// TwinCAT 3 PLC project RS485_HausBus
// ProgramVersion: 3.1.4024.0
// libraries:
//   Tc2_SerialCom, * (Beckhoff Automation GmbH)
//   Tc2_Standard, * (Beckhoff Automation GmbH)
//   Tc2_System, * (Beckhoff Automation GmbH)
//   Tc3_Module, * (Beckhoff Automation GmbH)
//   VisuDialogs, * (System)
//   VisuSymbols,3.5.10.0,System
// project tree:
//   DUTs/HausBus/BusTaster/ ST_BusTaster6F_Cnt.TcDUT, ST_BusTaster6F_Input.TcDUT, ST_BusTaster6F_Output.TcDUT
//   DUTs/HausBus/CYD/ ST_BusCYD6F_Input.TcDUT
//   DUTs/HausBus/RelaisModul/ ST_16Relais.TcDUT, ST_BusRelais16F_Cnt.TcDUT, ST_BusRelais16F_Input.TcDUT, ST_BusRelais16F_Output.TcDUT
//   DUTs/HausBus/Service/ ST_FiFoMaster_State.TcDUT, ST_RS485Startup_State.TcDUT (not stored)
//   DUTs/HausBus/ ST_HausBus_Ident.TcDUT
//   / GlobalTextList.TcGTLO, PlcTask.TcTTO, Visualisierungsmanager.TcVMO (not stored)
//   GVLs/ GVL.TcGVL
//   GVLs/RS485_HausBus/ GVL_HausBus_CONSTANT.TcGVL, GVL_HausBus_Devices.TcGVL, GVL_HausBus_Parameter.TcGVL, GVL_RS485FiFoSend.TcGVL, GVL_ServiceVisu.TcGVL
//   POUs/ RS485_COM_PRG.TcPOU
//   POUs/RS485_Hausbus_FB/CYD/ fb_CYDBus6F.TcPOU, fb_StringConvCYDService.TcPOU, fb_StringConvCYDWeb.TcPOU, fb_StringConvCYDWifi.TcPOU
//   POUs/RS485_Hausbus_FB/RS485 COM/FB/ fb_FilterArray.TcPOU
//   POUs/RS485_Hausbus_FB/RS485 COM/ fb_RS485ComCheck.TcPOU, fb_RS485IdScan.TcPOU, fb_RS485Ping.TcPOU
//   POUs/RS485_Hausbus_FB/RS485 COM/RS485_Master/ fb_RS485FiFoMaster.TcPOU, fb_RS485Startup.TcPOU
//   POUs/RS485_Hausbus_FB/BusTaster/ fb_StringConvTB6F.TcPOU, fb_TasterBus6F.TcPOU
//   POUs/RS485_Hausbus_FB/Events/ fb_BusRhdEvent.TcPOU, fb_BusTasterEvent.TcPOU, fb_BusPingEvent.TcPOU, fb_BusTempEvent.TcPOU, fb_BusBrsEvent.TcPOU
//   POUs/RS485_Hausbus_FB/RelaisModul/ fb_RelaisBus16F.TcPOU, fb_StringConvRB16F.TcPOU
//   VISUs/HausBus_RS485/ BusCYD6F_Frame.TcVIS, BusRelais16F_Frame.TcVIS, BusRS485Master_Frame.TcVIS, BusTatster6F_Frame.TcVIS, RS485HB_ServiceVISU.TcVIS
// real-time tasks:
//   TASK PlcTask: cycle T#1ms, priority 20, ADS port 350
// I/O:
//   DEVICE Gerät 2 (EtherCAT), AmsNetId 192.168.178.76.3.1
//     Box 1 (BK1120)
// variable links:
//   RS485_HausBus/RS485_HausBus Instance <-> Device 2 (EtherCAT)/Box 1 (BK1120)
//     PlcTask Inputs/.KL6041In/D[{0..21}] <-> Term 2 (KL6041)/Channel 1/Data In {0..21}  (22 links)
//     PlcTask Inputs/.KL6041In/Status <-> Term 2 (KL6041)/Channel 1/Status
//     PlcTask Inputs/.uiEtherCATStateBK1120_RS485COM <-> InfoData/State
//     PlcTask Inputs/.uiKBusStateBK1120_RS485COM <-> Inputs/CouplerState
//     PlcTask Outputs/.KL6041Out/Ctrl <-> Term 2 (KL6041)/Channel 1/Ctrl
//     PlcTask Outputs/.KL6041Out/D[{0..21}] <-> Term 2 (KL6041)/Channel 1/Data Out {0..21}  (22 links)

CONFIGURATION RS485_HausBus
    RESOURCE PLC ON TwinCAT3
        TASK PlcTask(INTERVAL := T#1ms, PRIORITY := 20);
        PROGRAM RS485_COM_PRG WITH PlcTask : RS485_COM_PRG;
    END_RESOURCE
END_CONFIGURATION

// ---- DUTs/HausBus/BusTaster/ST_BusTaster6F_Cnt.TcDUT
TYPE ST_BusTaster6F_Cnt :
STRUCT
	dwCntButtons    :ARRAY[1..6] OF DWORD;
END_STRUCT
END_TYPE

// ---- DUTs/HausBus/BusTaster/ST_BusTaster6F_Input.TcDUT
TYPE ST_BusTaster6F_Input :
STRUCT
	diID		:DINT;							(* Device ID ( Steht auf dem Aufkleber und wird zur Identifizierung im BUS benötigt)*)
	sName		:STRING;						(* Name des Tasters (zb- Wohnzimmer1 *)
	iLED      	:ARRAY[1..6] OF INT;     	  	(* gewünschter LED-Zustand (TRUE = 100 %)*)
	iLEDExt    	:ARRAY[1..6] OF INT;     	  	(* gewünschter LED-Zustand (TRUE = 100 %)*)
	iLEDBg		:INT;							(* gewünschte Hintergrundbeleuchtung *)
	bReset		:BOOL;							(* Reset des Tasters (Hardware) *)
	bExecute	:BOOL;							(* Aktivierung des Tasters *)
	bExtOutLED	:BOOL;							(* Verwendet die  Extra Ausgänge für LEDs / Mehr Busaulastung!  *)
END_STRUCT
END_TYPE

// ---- DUTs/HausBus/BusTaster/ST_BusTaster6F_Output.TcDUT
TYPE ST_BusTaster6F_Output :
STRUCT
	bButtons    :ARRAY[1..6] OF BOOL;       (*aktueller Tasterstatus (TRUE = gedrückt)*)
	bButtonsExt :ARRAY[1..6] OF BOOL;       (*aktueller Tasterstatus (TRUE = gedrückt)*)
	lrTemp		:LREAL;						(* Temperatur Sensor	*)
	lrRhd		:LREAL;						(* Luftfeuchtigkeit Sensor	*)
	lrBrs		:LREAL;						(* Helligkeit Sensor *)
	
	bCOM			:BOOL;					(*Zeigt die Kommunikation an *)
	bStartupDone	:BOOL;
	
	iState			:BOOL;
	sState			:STRING;
	bError			:BOOL;
END_STRUCT
END_TYPE

// ---- DUTs/HausBus/CYD/ST_BusCYD6F_Input.TcDUT
TYPE ST_BusCYD6F_Input :
STRUCT
	diID			:DINT;							(* Device ID ( Steht auf dem Aufkleber und wird zur Identifizierung im BUS benötigt)*)
	sName			:STRING;						(* Name des Tasters (zb- Wohnzimmer1 *)
	iLED      		:ARRAY[1..6] OF INT;     	  	(* gewünschter LED-Zustand (TRUE = 100 %)*)
	iLEDExt   	 	:ARRAY[1..6] OF INT;     	  	(* gewünschter LED-Zustand (TRUE = 100 %)*)
	iLEDBg			:INT;							(* gewünschte Hintergrundbeleuchtung *)
	
	
	bReset			:BOOL;							(* Reset des Tasters (Hardware) *)
	bExecute		:BOOL;							(* Aktivierung des Tasters *)
	bExtOutLED		:BOOL;							(* Verwendet die  Extra Ausgänge für LEDs / Mehr Busaulastung!  *)
	
	bServiceMode	:BOOL;
	bService		:BOOL;
	bWifi			:BOOL;
	bWebServer		:BOOL;
END_STRUCT
END_TYPE

// ---- DUTs/HausBus/RelaisModul/ST_16Relais.TcDUT
TYPE ST_16Relais :
STRUCT
	bOut	 : ARRAY[1..16] OF BOOL;
END_STRUCT
END_TYPE

// ---- DUTs/HausBus/RelaisModul/ST_BusRelais16F_Cnt.TcDUT
TYPE ST_BusRelais16F_Cnt :
STRUCT
	dwCntRelais    :ARRAY[1..16] OF DWORD;
END_STRUCT
END_TYPE

// ---- DUTs/HausBus/RelaisModul/ST_BusRelais16F_Input.TcDUT
TYPE ST_BusRelais16F_Input :
STRUCT
	diID		:DINT;							(* Device ID ( Steht auf dem Aufkleber und wird zur Identifizierung im BUS benötigt)*)
	sName		:STRING;						(* Name des Tasters (zb- Wohnzimmer1 *)
	bOut     	:ARRAY[1..16] OF BOOL;     	  	(* gewünschter Zustand (TRUE = An%)*)
	bReset		:BOOL;							(* Reset des Tasters (Hardware) *)
	bExecute	:BOOL;							(* Aktivierung des Tasters *)
END_STRUCT
END_TYPE

// ---- DUTs/HausBus/RelaisModul/ST_BusRelais16F_Output.TcDUT
TYPE ST_BusRelais16F_Output :
STRUCT
	bInputs		    :ARRAY[1..8] OF BOOL;       (*aktueller Tasterstatus (TRUE = gedrückt)*)
	bCOM			:BOOL;					(*Zeigt die Kommunikation an *)
	bStartupDone	:BOOL;
	
	iState			:BOOL;
	sState			:STRING;
	bError			:BOOL;
END_STRUCT
END_TYPE

// ---- DUTs/HausBus/Service/ST_FiFoMaster_State.TcDUT
TYPE ST_FiFoMaster_State :
STRUCT
	sReceiveString			:STRING(255);		
	lrBusAuslastung			:LREAL;
	bBusy					:BOOL;
	bDone					:BOOL;
	bError					:BOOL;
	iFiFoCount				:INT;
	iFiFoRow				:INT;
	sSendString				:STRING(255);
	sState					:STRING;
	
END_STRUCT
END_TYPE

// ---- DUTs/HausBus/ST_HausBus_Ident.TcDUT
TYPE ST_HausBus_Ident :
STRUCT
	diID			:DINT;							(* Device ID ( Steht auf dem Aufkleber und wird zur Identifizierung im BUS benötigt)*)
	sName			:STRING;						(* Name des Tasters (zb- Wohnzimmer1 *)	
	sPingIdent		:STRING :='TMP.1.gSTATUS'; 		(* Ping Identifiaktions String, wird bim Pingen gesendet  (Bei Taster = TMP.1.gSTATUS / Relais = OUT.210.rSTATUS / CYD= noch nicht definiert*)
	
END_STRUCT
END_TYPE

// ---- GVLs/GVL.TcGVL
{attribute 'Tc2GvlVarNames'}
VAR_GLOBAL

    KL6041In    					AT %I* : KL6inData22B; // Eingangsdaten von der Klemme
    KL6041Out 						AT %Q* : KL6outData22B; // Ausgangsdaten zur Klemme
	
	uiEtherCATStateBK1120_RS485COM	AT %I* : UINT;			// EtherCAT Status 
	uiKBusStateBK1120_RS485COM		AT %I* : UINT;			// Buskoppler Status
	
	fbTaster 						:ARRAY[1..cMaxBusTaster] OF fb_TasterBus6F;	
	fbRelais						:ARRAY[cMaxBusTaster+1..cMaxBusRelais+cMaxBusTaster+1] OF fb_RelaisBus16F;
END_VAR

// ---- GVLs/RS485_HausBus/GVL_HausBus_CONSTANT.TcGVL
{attribute 'Tc2GvlVarNames'}
VAR_GLOBAL CONSTANT
	cMaxBusTaster			:INT :=10;
	cMaxCYD					:INT :=2;
	cMaxBusRelais			:INT :=1;
	cMaxRS485CMDFiFo		:INT := 15;
	cMaxScanIDs				:INT :=50;
END_VAR

// ---- GVLs/RS485_HausBus/GVL_HausBus_Devices.TcGVL
{attribute 'Tc2GvlVarNames'}
VAR_GLOBAL
	stHBDeviceIdent					:ARRAY[1..cMaxRS485CMDFiFo] OF ST_HausBus_Ident;
	fbTasterHB6F 					:ARRAY[1..cMaxBusTaster] OF fb_TasterBus6F;	
	fbRelaisHB16F					:ARRAY[cMaxBusTaster+1..cMaxBusRelais+cMaxBusTaster+1] OF fb_RelaisBus16F;
	fbCYDHB6F 						:ARRAY[cMaxBusRelais+cMaxBusTaster+2..cMaxBusRelais+cMaxBusTaster+cMaxCYD+1] OF fb_CYDBus6F;	
END_VAR

// ---- GVLs/RS485_HausBus/GVL_HausBus_Parameter.TcGVL
{attribute 'Tc2GvlVarNames'}
VAR_GLOBAL
	
	(* Ping Abfrage *)
	bUseTasterPing						:BOOL := TRUE;			(* Schaltet die Ping empfangsüberprüfung ein um den Verbindungsstatus abzufragen*)
	cTimePingTimeTaster					:TIME := T#40S;			(* Ping Intervallzeit *)	(* Vorerst auf 5min gestellt, da die Taster Automatisch senden (Helligkeit/Luftfeuchtigkeit/Temp usw. *)
	cTimeReceiveTimeoutTaster			:TIME := T#200MS;		(* Ping Empfangs Timeout *)
	
	bUseRelaisPing						:BOOL := TRUE;			(* Schaltet die Ping empfangsüberprüfung ein um den Verbindungsstatus abzufragen*)
	cTimePingTimeRelais					:TIME := T#40S;			(* Ping Intervallzeit *)
	cTimeReceiveTimeoutRelais			:TIME := T#200MS;		(* Ping Empfangs Timeout *)
	
	bUseCYDPing							:BOOL := FALSE;			(* Schaltet die Ping empfangsüberprüfung ein um den Verbindungsstatus abzufragen*)
	cTimePingTimeCYD					:TIME := T#40S;			(* Ping Intervallzeit *)
	cTimeReceiveTimeoutCYD				:TIME := T#200MS;		(* Ping Empfangs Timeout *)
	
	(* FiFo Ping *)
	bUseFiFoPing						:BOOL := TRUE; 			(* Schaltet das Automatische Pingen vom FiFo Master ein, alle Geräte werden von dort aus angepingt *)
	cPingSendTimeFiFo					:TIME := T#19S;			(* Intervall Zeit, wann ein Ping vom FiFo gesendet werden soll an alle Devices *)
	
	(* Nicht verwendet *)
	cMaxPingTry							:INT  := 5;				(* Anzahl der Pingversuche *)
	
END_VAR

// ---- GVLs/RS485_HausBus/GVL_RS485FiFoSend.TcGVL
{attribute 'Tc2GvlVarNames'}
VAR_GLOBAL
	bSendDoneFiFo			:ARRAY[1..cMaxRS485CMDFiFo] OF BOOL;			(* Rückmeldung Aus dem FiFo Master Baustein, dass der Sendevorgang abgeschlossen ist *)
	sSendFiFo				:ARRAY[1..cMaxRS485CMDFiFo] OF STRING(255);		(* Zeile für den FiFo Master Baustein, von jedem einzelnen Busteilnehmer *)
END_VAR

// ---- GVLs/RS485_HausBus/GVL_ServiceVisu.TcGVL
{attribute 'Tc2GvlVarNames'}
VAR_GLOBAL
	iDeviceTasterVisu			:INT := 1;
	iDeviceRelaisVisu			:INT := cMaxBusTaster+1;
	iDeviceCYDVisu				:INT := cMaxBusTaster+cMaxBusRelais+1;
	
	bTasterServiceAktiv			:ARRAY[1..cMaxBusTaster] OF BOOL;
	bRelaisServiceAktiv			:ARRAY[cMaxBusTaster+1..cMaxBusTaster+cMaxBusRelais+1] OF BOOL;
	bCYDServiceAktiv			:ARRAY[cMaxBusRelais+cMaxBusTaster+2..cMaxBusRelais+cMaxBusTaster+cMaxCYD+1] OF BOOL;
	
	stTasterService				:ARRAY[1..cMaxBusTaster] OF ST_BusTaster6F_Input;
	stRelaisService				:ARRAY[cMaxBusTaster+1..cMaxBusTaster+cMaxBusRelais+1] OF ST_BusRelais16F_Input;
	stCYDService				:ARRAY[cMaxBusRelais+cMaxBusTaster+2..cMaxBusRelais+cMaxBusTaster+cMaxCYD+1] OF ST_BusCYD6F_Input;
END_VAR

// ---- POUs/RS485_COM_PRG.TcPOU
(*======================================================================================================================================*)
(*RS485_COM_PRG: Beispielhaftes Programm zum Steuern von HAus-Bus.de Komponenten über RS485 mit TwinCAT
					Achtung dieser POU muss als 1ms Task Aufgerufen werden um Ordnungsgemäß zu laufen *)
(*
Date          	| Version    	| created under        	| Author          	| Remark *)
(*====================================================================================================================================================*)
(*15/05/2025   	| 1.00      		| TC3		  		| N.Kersting       | first release *)
(*====================================================================================================================================================*)

PROGRAM RS485_COM_PRG
VAR  
     i,h,j						:INT;
	
	fbRS485Startup				:fb_RS485Startup;		(* Startup Parametrierung der Klemme/ RS485 Bus *)
	fbRS485SendCmdFiFo			:fb_RS485FiFoMaster;	(* Sende und Empfangs FiFo für RS485 *)
	fbLineControl 				:SerialLineControl;		(* Hält die Serielle Kommunikation Aufrecht *)
	
	fComBufferReset				:ClearComBuffer;		(* Löschen des SPS Internen Bufferinhalts *)
	
	rxBuffer 					:ComBuffer;				(* COM Buffer Empfangen *)
    txBuffer 					:ComBuffer;				(* COM Buffer Senden *)
	
	
END_VAR

(* IDs Setzen *)
ac00_HausBusIdRS485COM();
(* RS485 Klemmen Config *)
ac01_StartupRS485COM();

ACTION ac00_HausBusIdRS485COM:
(* Initialisierung der Gerätenamen *)
(* Achtung nur Beispiele *)
stHBDeviceIdent[1].sName	:=			'Wohnzimmer';
stHBDeviceIdent[1].diID	:=				5256;
stHBDeviceIdent[1].sPingIdent :=		'TMP.1.gSTATUS';

stHBDeviceIdent[2].sName	:=			'Test1';
stHBDeviceIdent[2].diID	:=				5269;
stHBDeviceIdent[2].sPingIdent :=		'TMP.1.gSTATUS';

stHBDeviceIdent[3].sName	:=			'Test2';
stHBDeviceIdent[3].diID	:=				1234;
stHBDeviceIdent[3].sPingIdent :=		'TMP.1.gSTATUS';

stHBDeviceIdent[4].sName	:=			'Test3';
stHBDeviceIdent[4].diID	:=				3333;
stHBDeviceIdent[4].sPingIdent :=		'TMP.1.gSTATUS';

stHBDeviceIdent[5].sName	:=			'Test4';
stHBDeviceIdent[5].diID	:=				4444;
stHBDeviceIdent[5].sPingIdent :=		'TMP.1.gSTATUS';

stHBDeviceIdent[6].sName	:=			'';
stHBDeviceIdent[6].diID	:=				0;
stHBDeviceIdent[6].sPingIdent :=		'TMP.1.gSTATUS';

stHBDeviceIdent[7].sName	:=			'';
stHBDeviceIdent[7].diID	:=				0;
stHBDeviceIdent[7].sPingIdent :=		'TMP.1.gSTATUS';

stHBDeviceIdent[8].sName	:=			'';
stHBDeviceIdent[8].diID	:=				0;
stHBDeviceIdent[8].sPingIdent :=		'TMP.1.gSTATUS';

stHBDeviceIdent[9].sName	:=			'';
stHBDeviceIdent[9].diID	:=				0;
stHBDeviceIdent[9].sPingIdent :=		'TMP.1.gSTATUS';

stHBDeviceIdent[10].sName	:=			'';
stHBDeviceIdent[10].diID	:=			0;
stHBDeviceIdent[10].sPingIdent :=		'TMP.1.gSTATUS';

stHBDeviceIdent[11].sName	:=			'Jalousie 1';
stHBDeviceIdent[11].diID	:=			5614;
stHBDeviceIdent[11].sPingIdent :=		'OUT.210.gSTATUS';

stHBDeviceIdent[12].sName	:=			'';
stHBDeviceIdent[12].diID	:=			0;
stHBDeviceIdent[12].sPingIdent :=		'OUT.210.gSTATUS';

stHBDeviceIdent[13].sName	:=			'CYD Test';
stHBDeviceIdent[13].diID	:=			5999;
stHBDeviceIdent[13].sPingIdent :=		'OUT.210.gSTATUS';
END_ACTION

ACTION ac01_StartupRS485COM:

(* Klemmen Startup, inkl Klemmenkonfiguration usw. *)
fbRS485Startup(
	I_bExecute:= 		TRUE, 
	I_bBusOK:= 			uiEtherCATStateBK1120_RS485COM = 8
						AND uiKBusStateBK1120_RS485COM = 0, 
	I_tStartupVerz:= 	T#5S, 
	IQ_InData:= 		KL6041In, 
	IQ_OutData:= 		KL6041Out, 
	Q_sState=> , 
	Q_bStartupDone=> , 
	Q_bError=> );

(* Aktivierung der Linecontrole erst wenn Startup erfolgt *)	
IF fbRS485Startup.Q_bStartupDone
THEN
	fbLineControl(
		Mode := 		ComSerialLineMode_t.SERIALLINEMODE_KL6_22B_STANDARD,
		pComIn := 		ADR(KL6041In),
		pComOut := 		ADR(KL6041Out),
		SizeComIn := 	UINT_TO_INT(SIZEOF(KL6041In)),
		RxBuffer := 	rxBuffer,
		TxBuffer := 	txBuffer );
				
	(* Relais *)
	ac10_HausBusRelaisRS485COM();
	(* Taster *)
	ac10_HausBusTasterRS485COM();
	(* CYD *)
	ac10_HausBusCYDRS485COM();
	
	
	(* Senden FiFo *)			
	fbRS485SendCmdFiFo(
		I_sSendCmdFiFo:= 		GVL_RS485FiFoSend.sSendFiFo, 
		I_stDeviceIdent :=		stHBDeviceIdent,
		I_bAutoPing:= 			bUseFiFoPing, 
		I_tAutoPingTime:= 		cPingSendTimeFiFo,		 
		I_bManuellMode:= 		, 
		I_sSendCmdManuell:= 	, 
		I_bSendManuell:= 		, 
		I_bExecute:= 			TRUE, 
		I_bBusBelastungstest:= 	, 
		I_bReset:= 				, 
		I_sStartZeichen:= 		, 
		I_sEndZeichen:= 		, 
		I_pTxBuffer:= 			ADR(txBuffer), 
		I_pRxBuffer:= 			ADR(rxBuffer), 
		Q_sReceiveString=> , 
		Q_lrBusAuslastung=> , 
		Q_bBusy=> , 
		Q_bDone=> , 
		Q_bError=> , 
		Q_sState=> , 
		Q_stStates=> );
		
ELSE
	(* Com Buffer zum Resetten *)
	fComBufferReset(Buffer:= rxBuffer);
	fComBufferReset(Buffer:= txBuffer);
END_IF
END_ACTION

ACTION ac10_HausBusCYDRS485COM:
(* Bustaster Aufrufe *)
FOR j := cMaxBusRelais+cMaxBusTaster+2 TO cMaxBusRelais+cMaxBusTaster+cMaxCYD+1 BY 1 DO
		
	fbCYDHB6F[j].I_stInput.sName :=	stHBDeviceIdent[j].sName;
	fbCYDHB6F[j].I_stInput.diID	:=	stHBDeviceIdent[j].diID;
	
	IF GVL_ServiceVisu.bCYDServiceAktiv[j]
	THEN
		fbCYDHB6F[j].I_stInput.iLED := GVL_ServiceVisu.stCYDService[j].iLED;
		fbCYDHB6F[j].I_stInput.iLEDBg := GVL_ServiceVisu.stCYDService[j].iLEDBg;
		fbCYDHB6F[j].I_stInput.iLEDExt := GVL_ServiceVisu.stCYDService[j].iLEDExt;
		fbCYDHB6F[j].I_stInput.bReset := GVL_ServiceVisu.stCYDService[j].bReset;
		fbCYDHB6F[j].I_stInput.bServiceMode := GVL_ServiceVisu.stCYDService[j].bServiceMode;
		fbCYDHB6F[j].I_stInput.bService := GVL_ServiceVisu.stCYDService[j].bService;
		fbCYDHB6F[j].I_stInput.bWifi := GVL_ServiceVisu.stCYDService[j].bWifi;
		fbCYDHB6F[j].I_stInput.bWebServer := GVL_ServiceVisu.stCYDService[j].bWebServer;
		
	END_IF
	
	stCYDService[j].sName :=	fbCYDHB6F[j].I_stInput.sName;
	stCYDService[j].diID :=		fbCYDHB6F[j].I_stInput.diID;
	
	fbCYDHB6F[j].I_stInput.bExecute := TRUE;
	fbCYDHB6F[j](
		I_FifoID :=			j,
		I_bPingStart:= 		TRUE , 	(* Taster Verzögert Pingen, damit weniger Busauslastung entsteht *)
		I_StringReceived:=	fbRS485SendCmdFiFo.Q_sReceiveString);
		
	(* Sendebefehle an FiFo Übergeben *)
	GVL_RS485FiFoSend.sSendFiFo[j] :=	fbCYDHB6F[j].Q_sFiFoSend;
END_FOR
END_ACTION

ACTION ac10_HausBusRelaisRS485COM:
(* BusRelais Aufrufe *)
FOR h := cMaxBusTaster +1 TO cMaxBusRelais+cMaxBusTaster+1 BY 1 DO (*cMaxBusTaster+1..cMaxBusRelais+cMaxBusTaster+1*)
		
	fbRelaisHB16F[h].I_stInput.sName :=	stHBDeviceIdent[h].sName;
	fbRelaisHB16F[h].I_stInput.diID	:=	stHBDeviceIdent[h].diID;
	
	IF GVL_ServiceVisu.bRelaisServiceAktiv[h]
	THEN
		fbRelaisHB16F[h].I_stInput.bOut := stRelaisService[h].bOut;
		fbRelaisHB16F[h].I_stInput.bReset := stRelaisService[h].bReset;
	END_IF
	
	stRelaisService[h].sName :=	fbRelaisHB16F[h].I_stInput.sName;
	stRelaisService[h].diID :=	fbRelaisHB16F[h].I_stInput.diID;
	
	fbRelaisHB16F[h].I_stInput.bExecute := TRUE;
	fbRelaisHB16F[h](
		I_FifoID :=			h,
		I_bPingStart:= 		TRUE,	(* Direkt Starten *)
		I_StringReceived:=	fbRS485SendCmdFiFo.Q_sReceiveString);
		
	(* Sendebefehle an FiFo Übergeben *)
	GVL_RS485FiFoSend.sSendFiFo[h] :=	fbRelaisHB16F[h].Q_sFiFoSend;	
END_FOR
END_ACTION

ACTION ac10_HausBusTasterRS485COM:
(* Bustaster Aufrufe *)
FOR i := 1 TO cMaxBusTaster BY 1 DO
			
	fbTasterHB6F[i].I_stInput.sName :=	stHBDeviceIdent[i].sName;
	fbTasterHB6F[i].I_stInput.diID	:=	stHBDeviceIdent[i].diID;
	
	IF GVL_ServiceVisu.bTasterServiceAktiv[i]
	THEN
		fbTasterHB6F[i].I_stInput.iLED := GVL_ServiceVisu.stTasterService[i].iLED;
		fbTasterHB6F[i].I_stInput.iLEDBg := GVL_ServiceVisu.stTasterService[i].iLEDBg;
		fbTasterHB6F[i].I_stInput.iLEDExt := GVL_ServiceVisu.stTasterService[i].iLEDExt;
		fbTasterHB6F[i].I_stInput.bReset := GVL_ServiceVisu.stTasterService[i].bReset;
	END_IF
	
	stTasterService[i].sName :=	fbTasterHB6F[i].I_stInput.sName;
	stTasterService[i].diID :=	fbTasterHB6F[i].I_stInput.diID;
	
	fbTasterHB6F[i].I_stInput.bExecute := TRUE;
	fbTasterHB6F[i](
		I_FifoID :=			i,
		I_bPingStart:= 		TRUE , 	(* Taster Verzögert Pingen, damit weniger Busauslastung entsteht *)
		I_StringReceived:=	fbRS485SendCmdFiFo.Q_sReceiveString);
		
	(* Sendebefehle an FiFo Übergeben *)
	GVL_RS485FiFoSend.sSendFiFo[i] :=	fbTasterHB6F[i].Q_sFiFoSend;
END_FOR
END_ACTION

END_PROGRAM

// ---- POUs/RS485_Hausbus_FB/RS485 COM/RS485_Master/fb_RS485Startup.TcPOU
(*======================================================================================================================================*)
(*fb_RS485Startup:	Einfacher Baustein um die Hardware für die RS485 Haus-Bus vorzubereiten*)
(*
Date          	| Version    	| created under        	| Author          	| Remark *)
(*====================================================================================================================================================*)
(*13/05/2025   	| 1.00      		| TC3		  		| N.Kersting       | first release *)
(*====================================================================================================================================================*)
FUNCTION_BLOCK fb_RS485Startup
VAR_INPUT
	I_bExecute						:BOOL;
	I_bBusOK						:BOOL;
	I_tStartupVerz					:TIME := T#2S;	(* Startup verzögert ausführen *)
END_VAR
VAR_IN_OUT
	IQ_InData	 					:KL6inData22B;
    IQ_OutData						:KL6outData22B;
END_VAR
VAR_OUTPUT
	Q_sState						:STRING;
	Q_bStartupDone					:BOOL;
	Q_bError						:BOOL;
	Q_stStates						:ST_RS485Startup_State;
END_VAR
VAR
	udBaudrate						:UDINT := 57600;
	byDataBits						:BYTE := 8;
	byStopBits						:BYTE := 1;
	
	tonStartupVerz					:ton;
	fbSerialComReset				:ComReset;
	fComBufferReset					:ClearComBuffer;
	fbSerialConfig 					:KL6Configuration;  // Terminal-Konfiguration (Baud, Parität etc.)
	iStepStartup					:INT;
END_VAR

tonStartupVerz(
	PT :=	I_tStartupVerz);
	
CASE iStepStartup OF 
(*=========================================================================*)
0:	IF NOT Q_bError
		AND I_bBusOK
	THEN
		Q_sState := 'INIT';
	ELSIF
		NOT I_bBusOK
	THEN
		Q_bError := TRUE;
		Q_sState := 'Busverbindung nicht Ok';
	END_IF
	
	tonStartupVerz.IN := FALSE;
	
	fbSerialComReset(
		Execute:= 		FALSE);
		
	fbSerialConfig(
		Execute:= 		FALSE);
		
	IF I_bExecute
		AND I_bBusOK
	THEN
		Q_bStartupDone := FALSE;
		iStepStartup := iStepStartup+1;
	END_IF

(*=========================================================================*)
1:	Q_sState := 'Warten auf Verzögerung';
	tonStartupVerz.IN := TRUE; 
	
	IF tonStartupVerz.Q
	THEN
		iStepStartup := iStepStartup+1;
	END_IF
	
(*=========================================================================*)
2:	Q_sState := 'Serielle Klemme Konfigurieren mit Haus-Bus Vorgaben';	
	
	fbSerialConfig(
		Execute:= 		TRUE, 
		Mode:= 			ComSerialLineMode_t.SERIALLINEMODE_KL6_22B_STANDARD,		 
		Baudrate:= 		udBaudrate, 
		NoDatabits:= 	byDataBits, 
		Parity:= 		ComParity_t.PARITY_EVEN,	 
		Stopbits:= 		byStopBits, 
		Handshake:= 	RS485_HALFDUPLEX, 
		ContinousMode:= , 
		pComIn := 		ADR(IQ_InData), 
		pComOut := 		ADR(IQ_OutData), 
		SizeComIn := 	SIZEOF(IQ_InData),
		Done=> , 
		Busy=> , 
		Error=> , 
		ErrorId=> );
	
	IF fbSerialConfig.Done
	THEN
		fbSerialConfig(
			Execute:= 		FALSE); 
			
		iStepStartup := 3;
	ELSIF
		fbSerialConfig.Error
	THEN
		Q_sState := 'Error fbSerialConfig ID: ';
		Q_sState := CONCAT(Q_sState,INT_TO_STRING(fbSerialConfig.ErrorID));
		iStepStartup := -2;	//Error
	END_IF

(*=========================================================================*)
3:	Q_sState := 'Serielle Klemme Reset Auführen';	
		
	fbSerialComReset(
		Execute:= 		TRUE, 
		pComIn := 		ADR(IQ_InData), 
		pComOut := 		ADR(IQ_OutData), 
		SizeComIn := 	SIZEOF(IQ_InData),
		Done=> , 
		Busy=> , 
		Error=> , 
		ErrorID=> );	
		
	IF fbSerialComReset.Done
	THEN
		iStepStartup := 999;
	ELSIF
		fbSerialComReset.Error
	THEN
		Q_sState := 'Error fbSerialComReset ID: ';
		Q_sState := CONCAT(Q_sState,INT_TO_STRING(fbSerialComReset.ErrorID));
		iStepStartup := -3;	//Error
	END_IF
	
(*=========================================================================*)
999:Q_sState := 'Startup Ausgeführt!';	
	Q_bStartupDone := TRUE;
	Q_bError := FALSE;
	
	IF NOT I_bBusOK
	THEN
		Q_bStartupDone := FALSE;
		iStepStartup := 0;
	END_IF

ELSE
	(* ERROR *)
	Q_bError := TRUE;
	iStepStartup := 0;
END_CASE

(* StatusStruktur für Visu *)
Q_stStates.bBusOk				:=	I_bBusOK;
Q_stStates.bStartupDone			:=	Q_bStartupDone;
Q_stStates.bStartupError		:=	Q_bError;
Q_stStates.sStartupState		:=	Q_sState;

END_FUNCTION_BLOCK

// ---- POUs/RS485_Hausbus_FB/RS485 COM/RS485_Master/fb_RS485FiFoMaster.TcPOU
(*======================================================================================================================================*)
(*fb_RS485FiFoMaster:	Einfaches Senden eines Telegrams über RS485*)
(*
Date          	| Version    	| created under        	| Author          	| Remark *)
(*====================================================================================================================================================*)
(*10/05/2025   	| 1.00      		| TC3		  		| N.Kersting       | first release *)
(*10/05/2025   	| 1.01      		| TC3		  		| N.Kersting       | Nun wird der Empfang auch mit Implementiert  *)
(*13/05/2025   	| 1.02      		| TC3		  		| N.Kersting       | Busbelastungstest Implementiert - Sendet Durchgehend Strings *)
(*14/05/2025   	| 1.03      		| TC3		  		| N.Kersting       | Busauslastung direkt Implementiert *)
(*27/05/2025   	| 1.04      		| TC3		  		| N.Kersting       | Neuen Manuell Mode implementiert um einen Manuell generierten String allein zu Senden *)
(*28/05/2025   	| 1.05      		| TC3		  		| N.Kersting       | Neue Automatisch Ping Funktion hinzugefügt & Wichtiger Bugfix *)
(*02/06/2025   	| 2.00      		| TC3		  		| N.Kersting       | Neue Verbesserte Collision Detection, verhindert, dass Senden bei gefülltem Epmfangspuffer *)
(*03/06/2025   	| 2.01      		| TC3		  		| N.Kersting       | Collision Detection nun aufgeeilt in Empfang und Senden *)
(*03/06/2025   	| 2.02      		| TC3		  		| N.Kersting       | Neue Bus Scan Funktion Implementiert, Scannt alle Teilnehmer Ids im Bus (nur im Manuell Mode verfügbar) *)
(*====================================================================================================================================================*)
FUNCTION_BLOCK fb_RS485FiFoMaster
VAR_INPUT
	I_sSendCmdFiFo				:ARRAY[1..cMaxRS485CMDFiFo] OF STRING(255);
	I_stDeviceIdent				:ARRAY[1..cMaxRS485CMDFiFo] OF ST_HausBus_Ident;	(* Um Zyklisch einzelnt anzupingen *)
	
	I_bAutoPing					:BOOL;												(* Wenn Aktiv wird Zyklisch Automatisch ein Ping gesendet, welcher von den einzelnen Kommunikationsbausteinen ausgewertet werden kann *)
	I_tAutoPingTime				:TIME :=T#10S;										(* Die Intervallzeit, Bis ein Auto Ping gesendet wird *)
	
	I_bManuellMode				:BOOL := FALSE;
	I_bSearchMode				:BOOL := FALSE;
	I_sSendCmdManuell			:STRING(255);
	I_bSendManuell				:BOOL;
	I_bExecute					:BOOL := TRUE;
	I_bBusBelastungstest		:BOOL;
	I_bReset					:BOOL;
	I_sStartZeichen				:BYTE := 16#FD;										(* Startzeichen Präfix *)
	I_sEndZeichen				:BYTE := 16#FE;										(* Endzeichen Suffix *)
	I_pTxBuffer					:POINTER TO ComBuffer; 								(* Zeiger auf TX-Buffer*)
	I_pRxBuffer   				:POINTER TO ComBuffer;  							(* Zeiger auf RX-Buffer*)
END_VAR
VAR_OUTPUT
	Q_sReceiveString			:STRING(255);		
	Q_lrBusAuslastung			:LREAL;
	Q_bBusy						:BOOL;
	Q_bDone						:BOOL;
	Q_bError					:BOOL;
	Q_sState					:STRING;
	Q_stStates					:ST_FiFoMaster_State;
END_VAR
VAR
(*==========================================================================================================*)
(* Parameter *)
(*==========================================================================================================*)
	bActivateSend				:BOOL := TRUE;					(* Aktiviert das Senden von Nachrichten *)
	bActivateReceive			:BOOL := TRUE;					(* Aktiviert das Empfangen von Nachrichten *)
	
	bUseRXCollisionDetection	:BOOL := TRUE;					(* Aktiviert die Empfangs Kollisions Überprüfung *)
	bUseTXCollisionDetection	:BOOL := FALSE;					(* Aktiviert die Sende Kollisions Überprüfung *)
	tVerzCollisionDetect		:TIME := T#100MS;				(* Zeit, die zum Empfangen bleibt *)
(*==========================================================================================================*)	
	bRXCollisionDetected		:BOOL;
	bTXCollisionDetected		:BOOL;
	bCollisionFree				:BOOL;	
(*==========================================================================================================*)		
	bFirstCycle					:BOOL := TRUE;
	bStringSend					:BOOL := FALSE;
	bBusBelastungstest			:BOOL := FALSE;
	bBusAuslastung				:BOOL := TRUE;
	bPingStart					:BOOL;
	bBusyMem					:BOOL;
(*==========================================================================================================*)	
	sReceivedMEMString			:STRING(255);
	sReceivedString				:STRING(255);
	sStep						:STRING;
	sString						:STRING(255);
	sStringSend					:STRING(255);
(*==========================================================================================================*)		
	iStep						:INT;
	iStepReceive				:INT;
	iMaxBufferBlocking			:INT := 20;
	icntError					:INT;
	iFiFoRow					:INT := 1;
	icntFiFo					:INT;
	i,h							:INT;
	iStepFiFo					:INT;
(*==========================================================================================================*)		

	tonCollisionFree			:ton;	
	tonTimeout					:ton;
	tonPingIntervall			:ton;
	tonSend						:ton;
(*==========================================================================================================*)		
	rTrigSendManuell			:r_Trig;
	rTrigSendSearchMode			:r_trig;
	fbSend     					:SendString255;
	fbReceive   				:ReceiveString255;
	fbBusAuslastung				:fb_FilterArray;
	
	fbRS485Search				:fb_RS485IdScan;
END_VAR

(*============================================================================================*)
(* Laufzeit fehler *)
tonTimeout(
	PT:=T#1S);
	
(*============================================================================================*)		
(* Collision detection, soll verhinddern, dass nicht gesendet wird, wenn Daten im Empfangsüpuffer sind *)
(* Receive Collision Dectetion *)
bRXCollisionDetected :=	(I_pRxBuffer^.Count > INT_TO_UINT(iMaxBufferBlocking) 
						OR I_pRxBuffer^.FreeByte < (301 -INT_TO_UINT(iMaxBufferBlocking))
						OR I_pRxBuffer^.blocked
						OR I_pRxBuffer^.Error <> 0
						OR fbReceive.StringReceived
						(*OR sReceivedString <> ''*))
						AND bUseRXCollisionDetection;
						
(* Transmit Collision Detection *)
bTXCollisionDetected :=	(I_pTxBuffer^.Count > INT_TO_UINT(iMaxBufferBlocking) 
						OR I_pTxBuffer^.FreeByte < (301 -INT_TO_UINT(iMaxBufferBlocking))
						OR I_pTxBuffer^.blocked
						OR I_pTxBuffer^.Error <> 0)
						AND bUseTXCollisionDetection;
						
(* Collision Detection Verzögern *)						
tonCollisionFree(
	IN := 	NOT bRXCollisionDetected
			AND NOT bTXCollisionDetected,
	PT := 	tVerzCollisionDetect,
	Q =>	bCollisionFree);

(*============================================================================================*)	
(* Ping Intervall Timer *)		
tonPingIntervall(
	IN := I_bAutoPing
			AND NOT bPingStart,
	PT := I_tAutoPingTime);
	
(*============================================================================================*)	
(* Busbelastungstest *)	
bBusBelastungstest := I_bBusBelastungstest;
sReceivedMEMString:='';

(*============================================================================================*)	
(* Anzahl der gefüllten FiFo Zeilen *)
icntFiFo := 0;
FOR i := 1 TO cMaxRS485CMDFiFo BY 1 DO 
	IF (I_sSendCmdFiFo[i]<> '')
	THEN
		icntFiFo := icntFiFo +1;
	END_IF
END_FOR

(*============================================================================================*)	
(* Manuelles Senden *)
rTrigSendManuell(
	CLK := I_bSendManuell);

(*============================================================================================*)
CASE iStepFiFo OF
-1:	sStep := 'FiFo INIT';
	bFirstCycle := FALSE;
	Q_bBusy := FALSE;
	bPingStart := FALSE;
	iFiFoRow := 1;
	
	FOR h := 1 TO cMaxRS485CMDFiFo BY 1 DO
		GVL_RS485FiFoSend.bSendDoneFiFo[h] :=TRUE;
	END_FOR
	
	iStepFiFo := 0;

(*============================================================================================*)
0:	sStep := 'Warten, dass FiFo gefüllt wird';
	iFiFoRow := 1;
	bStringSend := FALSE;
	Q_bBusy := FALSE;
			
	(* Wenn die Intervall Zeit abgelaufen ist Ping Start setzen *)
	IF tonPingIntervall.Q
	THEN
		bPingStart := TRUE;
	END_IF
	
	IF (icntFiFo > 0
		OR  bBusBelastungstest
		OR I_bManuellMode)
		AND NOT bFirstCycle
		AND NOT bPingStart
		AND bCollisionFree
	THEN
		Q_bBusy := TRUE;
		iStepFiFo := 1;
	ELSIF
		bFirstCycle
	THEN
		iStepFiFo := -1;
	ELSIF
		bPingStart
		AND NOT bFirstCycle
		AND bCollisionFree
	THEN
		iStepFiFo := 10;	(* Ping senden *)
	END_IF
	
(*============================================================================================*)	
1:	sStep := 'Prüfen ob STRING in FiFo Zeile gefüllt*';
	
	IF I_bSearchMode
	THEN
		sStep :=fbRS485Search.Q_sState;
	END_IF
	
	(* Manueller Modus *)
	IF I_bManuellMode
	THEN
		(* Prüfen ob in der Zeile etwas steht *)
		IF I_sSendCmdManuell <>''
			AND rTrigSendManuell.Q
			AND NOT I_bSearchMode
		THEN
			IF bCollisionFree
			THEN
				sString :=	I_sSendCmdManuell; 
				bStringSend := TRUE;
				Q_bDone := FALSE;
				Q_bError := FALSE;
				iStepFiFo := iStepFiFo+1;
			END_IF
		END_IF
		(* Prüfen ob in der Zeile etwas steht *)
		IF I_bSearchMode
			AND fbRS485Search.Q_bSend
		THEN
			IF bCollisionFree
			THEN
				sString :=	fbRS485Search.Q_sSearchString; 
				bStringSend := TRUE;
				Q_bDone := FALSE;
				Q_bError := FALSE;
				iStepFiFo := iStepFiFo+1;
			END_IF
		END_IF
	ELSE
		(* Prüfen ob in der ausgewählten Zeile etwas steht *)
		sStringSend :=	I_sSendCmdFiFo[iFiFoRow]; 
		IF I_sSendCmdFiFo[iFiFoRow] = ''
		THEN
			IF iFiFoRow < cMaxRS485CMDFiFo
			THEN
				iFiFoRow := iFiFoRow+1; (* Nächste Zeile, bis etwas drin Steht *)
			ELSE
				IF bBusBelastungstest
				THEN
					sStringSend :=	CONCAT(F_ToCHR(I_sStartZeichen),'ServiceTOOL-BUSBELASTUNGSTEST-BURSTFIREMODE');
					sStringSend :=	CONCAT(sStringSend,F_ToCHR(I_sEndZeichen));
					(* Senden *)
					
					IF  bCollisionFree
					THEN
						sStep := 'Prüfe ob Senden noch aktiv ist';
						bStringSend := TRUE;
						sString :=	sStringSend;
						Q_bDone := FALSE;
						Q_bError := FALSE;
						iStepFiFo := iStepFiFo+1;
					END_IF
				ELSE
					iStepFiFo := 0;	(* Alle Zeilen Abgearbeitet *)
				END_IF
			END_IF
		ELSE
		(* Senden *)
		GVL_RS485FiFoSend.bSendDoneFiFo[iFiFoRow] :=FALSE;
		
			IF bCollisionFree
			THEN
				sStep := 'Prüfe ob Senden noch aktiv ist';
				bStringSend := TRUE;
				sString :=	sStringSend;
				Q_bDone := FALSE;
				Q_bError := FALSE;
				iStepFiFo := iStepFiFo+1;
			END_IF
		END_IF
	END_IF
	
(*============================================================================================*)		
2:	sStep := 'Starte Senden';
	Q_bBusy := TRUE;
	tonTimeout.IN := fbSend.Busy;
	
	IF NOT fbSend.Busy
		AND NOT fbReceive.StringReceived
	THEN
		sString := '';
		tonSend.IN := FALSE;
		bStringSend := FALSE;
		iStepFiFo := iStepFiFo+1;
	ELSIF
		(fbSend.Error >0)
		AND NOT (fbSend.Error = 2)
	THEN
		sStep := CONCAT('ERROR-',sStep);
		sStep := CONCAT(sStep,'- ');
		sStep := CONCAT(sStep,INT_TO_STRING(fbSend.Error));
		iStepFiFo := -2;
	ELSIF
		tonTimeout.Q
	THEN
		sStep := CONCAT('ERROR- Timeout',sStep);
		iStepFiFo := -2;
	END_IF
	
(*============================================================================================*)		
3:	(* Senden*)		
	GVL_RS485FiFoSend.bSendDoneFiFo[iFiFoRow] :=TRUE;
	
	IF iFiFoRow < cMaxRS485CMDFiFo
		AND NOT I_bSearchMode
	THEN
		iFiFoRow := iFiFoRow+1;
		iStepFiFo := 1;
	ELSE
		Q_bDone := TRUE;
		
		IF (NOT fbRS485Search.Q_bSend
			AND I_bSearchMode)
			OR NOT I_bSearchMode
		THEN
			iStepFiFo := 0;
		END_IF
		
	END_IF
	
(*============================================================================================*)	
(* Ping Senden Ablauf *)
(*============================================================================================*)	
10:	sStep := 'Sende Ping*';
	
	(* Ping String erstellen *)
	sStringSend:=	CONCAT(F_ToCHR(I_sStartZeichen),DINT_TO_STRING(I_stDeviceIdent[iFiFoRow].diID));
	sStringSend :=	CONCAT(sStringSend,'.');
	sStringSend :=	CONCAT(sStringSend ,I_stDeviceIdent[iFiFoRow].sPingIdent); 
	sStringSend :=	CONCAT(sStringSend,F_ToCHR(I_sEndZeichen));
	
	IF I_stDeviceIdent[iFiFoRow].sPingIdent = ''
		OR I_stDeviceIdent[iFiFoRow].diID = 0
	THEN
		IF iFiFoRow < cMaxRS485CMDFiFo
		THEN
			iFiFoRow := iFiFoRow+1; (* Nächste Zeile, bis etwas drin Steht *)
		ELSE
			bPingStart := FALSE;
			iStepFiFo := 0;	(* Alle Zeilen Abgearbeitet *)
		END_IF
	ELSE
	(* Senden *)	
		IF bCollisionFree
		THEN
			sStep := 'Prüfe ob Senden noch aktiv ist';
			bStringSend := TRUE;
			sString :=	sStringSend;
			Q_bDone := FALSE;
			Q_bError := FALSE;
			iStepFiFo := iStepFiFo+1;
		END_IF
	END_IF
	
(*============================================================================================*)		
11:	sStep := 'Starte Senden';
	Q_bBusy := TRUE;
	tonTimeout.IN := fbSend.Busy;
	
	IF NOT fbSend.Busy
		AND NOT fbReceive.StringReceived
	THEN
		tonSend.IN := FALSE;
		bStringSend := FALSE;
		iStepFiFo := iStepFiFo+1;
	ELSIF
		(fbSend.Error >0)
		AND NOT (fbSend.Error = 2)
	THEN
		sStep := CONCAT('ERROR-',sStep);
		sStep := CONCAT(sStep,'- ');
		sStep := CONCAT(sStep,INT_TO_STRING(fbSend.Error));
		iStepFiFo := -2;
	ELSIF
		tonTimeout.Q
	THEN
		sStep := CONCAT('ERROR- Timeout',sStep);
		iStepFiFo := -2;
	END_IF
	
(*============================================================================================*)		
12:	(* Senden*)		

	IF iFiFoRow < cMaxRS485CMDFiFo
	THEN
		iFiFoRow := iFiFoRow+1;
		iStepFiFo := 10;
	ELSE
		bPingStart := FALSE;
		iStepFiFo := 0;
	END_IF
	
ELSE
(*============================================================================================*)
	Q_bError := TRUE;
	Q_bBusy := FALSE;
	bBusyMem := FALSE;
	tonTimeout.IN := FALSE;
	
	IF I_bReset
	THEN
		iStepFiFo := 0;
	END_IF
END_CASE

(*============================================================================================*)	
(* Nur Senden, wenn nicht Empfangen wird *)
IF bStringSend
THEN
	IF bActivateSend
	THEN
		(* Senden *)
		fbSend(
			SendString:= 	sString,
			TXbuffer:= 		I_pTxBuffer^);
	END_IF
	
ELSE
	IF bActivateReceive
	THEN
		(* Empfangen *)
		ac00_Receive();
	END_IF
END_IF

(*============================================================================================*)	
(* Empfangsmerker 0 Setzen am ende Eines Zyklus *)
Q_sReceiveString := sReceivedMEMString;

(*============================================================================================*)	
(* Busauslastung tracken*)
ac99_Diagnose();

(*============================================================================================*)	
(* StatusStruktur für Visu *)
Q_sState :=	sStep;
Q_stStates.bBusy				:=	Q_bBusy;
Q_stStates.bDone				:=	Q_bDone;
Q_stStates.bError				:=	Q_bError;
Q_stStates.iFiFoCount			:=	icntFiFo;
Q_stStates.iFiFoRow				:=	iFiFoRow;
Q_stStates.lrBusAuslastung		:=	Q_lrBusAuslastung;
Q_stStates.sReceiveString 		:=	Q_sReceiveString;
Q_stStates.sSendString 			:=	sString;
Q_stStates.sState 				:=	Q_sState;

ACTION ac00_Receive:
(*============================================================================================*)	
(* Empfangen *)

CASE iStepReceive OF		
0:	fbReceive(
		Prefix := 			F_ToCHR(I_sStartZeichen),
		Suffix := 			F_ToCHR(I_sEndZeichen),
		Timeout:= , 
		Reset:= , 
		StringReceived=> , 
		Busy=> , 
		Error=> , 
		RxTimeout=> , 
		ReceivedString:= 	sReceivedString, 
		RXbuffer:= 			I_pRxBuffer^);
		
	IF fbReceive.StringReceived
	THEN
		iStepReceive := 1;
		sReceivedMEMString := sReceivedString;
	END_IF
	
1:	sReceivedString := '';
	iStepReceive := 0;
	
END_CASE
END_ACTION

ACTION ac99_Diagnose:
(*============================================================================================*)	
(* Busauslastung Prüfen *)

fbBusAuslastung(
	I_bExcecute:= 	bBusAuslastung, 
	I_nWert:= 		UINT_TO_LREAL(I_pTxBuffer^.Count), 
	I_nFilterWert:= 50, 
	Q_nFilter=> 	Q_lrBusAuslastung);
	
	
fbRS485Search(
	I_bStartSearch:= 	I_bSearchMode, 
	I_diStartID:= , 
	I_diMaxID:= , 
	I_sStartZeichen:= 	I_sStartZeichen, 
	I_sEndZeichen:= 	I_sEndZeichen, 
	I_tWait:= , 
	I_StringReceived:= 	sReceivedMEMString, 
	Q_bSend=> , 
	Q_sSearchString=> );
END_ACTION

END_FUNCTION_BLOCK

// ---- POUs/RS485_Hausbus_FB/RS485 COM/FB/fb_FilterArray.TcPOU
(*======================================================================================================================================*)
(* Dieser Baustein Filtert eine Lreal Variable durch bildung eines Mittelwerts
(*======================================================================================================================================*)						

Date          		| Version    		| created under        		| Author          		| Remark *)
(*======================================================================================================================================*)
(*´10/07/2024   	| 1.00      			| TC2			  		| N.Kersting       	| first release *)
(*´15/07/2024   	| 1.01      			| TC2			  		| N.Kersting       	| Filterung nun Variabel einstellbar *)
(*======================================================================================================================================*)
FUNCTION_BLOCK fb_FilterArray
VAR_INPUT
	I_bExcecute	:BOOL;
	I_nWert		:LREAL;
	I_nFilterWert	:INT	:= 10;
END_VAR
VAR_OUTPUT
	Q_nFilter		:LREAL;
END_VAR
VAR
	i	:INT;
	nWertArray	:ARRAY [0..50] OF LREAL;
END_VAR

IF I_bExcecute THEN
   (* // Verschieben der Werte im Array*)
    FOR i := I_nFilterWert - 1 TO 1 BY -1 DO
        nWertArray[i] := nWertArray[i - 1];
    END_FOR

   (* // Neuen Wert einfügen	*)
    nWertArray[0] := I_nWert;

  (*  // Berechnung des gefilterten Wertes*)
    Q_nFilter := 0;
    FOR i := 0 TO I_nFilterWert - 1 DO
        Q_nFilter := Q_nFilter + nWertArray[i];
    END_FOR
    Q_nFilter := Q_nFilter / I_nFilterWert;

ELSE
  (*  // Initialisieren des Arrays*)
    FOR i := 0 TO 10 DO
        nWertArray[i] := 0;
    END_FOR
    Q_nFilter := 0;
END_IF

// ---- POUs/RS485_Hausbus_FB/RS485 COM/fb_RS485IdScan.TcPOU
(*======================================================================================================================================*)
(*fb_RS485Search:	Suchfunktion um Automatisch alle ID's im Bus zu Scannen*)
(*
Date          	| Version    	| created under        	| Author          	| Remark *)
(*====================================================================================================================================================*)
(*03/06/2025   	| 1.00      		| TC3		  		| N.Kersting       | first release *)
(*====================================================================================================================================================*)
FUNCTION_BLOCK fb_RS485IdScan
VAR_INPUT
	I_bStartSearch		:BOOL;
	I_diStartID			:DINT	:= 5000;
	I_diMaxID			:DINT	:= 6000;
	I_sStartZeichen		:BYTE := 16#FD;										(* Startzeichen Präfix *)
	I_sEndZeichen		:BYTE := 16#FE;										(* Endzeichen Suffix *)
	I_tWait				:TIME := T#300MS;
	I_StringReceived	:STRING(255);
END_VAR
VAR_OUTPUT
	Q_bSend				:BOOL;
	Q_sSearchString		:STRING(255);
	Q_iCnt				:INT;
	Q_sState			:STRING;
	Q_sIDList			:ARRAY[1..cMaxScanIDs] OF DINT;
END_VAR
VAR
	i					:INT;
	iArrIdx				:INT := 1;
	fbPingEvent			:fb_BusPingEvent;
	diActId				:DINT;
	iStep				:INT;
	tonWait				:ton;
	rTrigSearch			:r_trig;
END_VAR


tonWait(
	PT := I_tWait);
	
rTrigSearch(CLK:= I_bStartSearch, Q=> );

IF NOT I_bStartSearch
THEN
	iStep := 0;
END_IF
	
CASE iStep OF
(*=========================================================================*)
0:	Q_sState := 'INIT';
	tonWait.IN := FALSE;
	Q_bSend := FALSE;
	diActId := I_diStartID;
	Q_sSearchString := '';
	iArrIdx := 1;
	Q_iCnt := 0;
	
	IF rTrigSearch.Q
		AND I_diStartID >0
		AND I_diMaxID >0
	THEN
		FOR i := 1 TO cMaxScanIDs BY 1 DO 
			Q_sIDList[i] := 0;
		END_FOR
		
		iStep := iStep +1;
	END_IF
	
(*=========================================================================*)
1:	Q_bSend := FALSE;
	tonWait.IN := FALSE;
	
	IF diActId <= I_diMaxID
	THEN		
		iStep := iStep +1;
	ELSE
		iStep := 0;
	END_IF
	
(*=========================================================================*)
2:	Q_sSearchString := CONCAT(F_ToCHR(I_sStartZeichen),DINT_TO_STRING(diActId));
	Q_sSearchString := CONCAT(Q_sSearchString,'.TMP.1.gSTATUS');
	Q_sSearchString := CONCAT(Q_sSearchString,F_ToCHR(I_sEndZeichen));
	Q_sSearchString := CONCAT(Q_sSearchString,F_ToCHR(I_sStartZeichen));
	Q_sSearchString := CONCAT(Q_sSearchString,DINT_TO_STRING(diActId));
	Q_sSearchString := CONCAT(Q_sSearchString,'.OUT.210.gSTATUS');
	Q_sSearchString := CONCAT(Q_sSearchString,F_ToCHR(I_sEndZeichen));
	
	iStep := iStep +1;
	
(*=========================================================================*)
3:	Q_sState := 'Suchen Aktiv';
	tonWait.IN := TRUE;
	Q_bSend := TRUE;
	
	fbPingEvent(
		I_sID:= 				DINT_TO_STRING(diActId), 
		I_sReceivedString:= 	I_StringReceived, 
		I_bReset:= ,
		Q_bOut=> );
		
	IF fbPingEvent.Q_bOut
	THEN
		Q_bSend := FALSE;
		iStep := iStep +1;
	ELSIF
		tonWait.Q
	THEN
		Q_bSend := FALSE;
		IF diActId <I_diMaxID
		THEN
			diActId := diActId +1;
			iStep := 1; (* nächsten Teilnehmer Suchen *)
		ELSE
			iStep := 6;	(* Scan Fertig *)
		END_IF
	END_IF
	
(*=========================================================================*)
4:	(* Teilnehmer gefunden ! *)
	Q_sState := 'Teilnehmer gefunden!';
	tonWait.IN := FALSE;	
	Q_bSend := FALSE;
	Q_sIDList[iArrIdx] := diActId;
	
	IF diActId <I_diMaxID
	THEN
		IF iArrIdx < cMaxScanIDs 
		THEN
			diActId := diActId +1;
			iArrIdx := iArrIdx +1;
			iStep := 1; (* nächsten Teilnehmer Suchen *)
		ELSE
			iStep := 5;
		END_IF
	ELSE
		iStep := 6;	(* Scan Fertig *)
	END_IF
	
(*=========================================================================*)
5:	(* Liste Voll! *)
	Q_sState := 'Liste Voll!';
	
(*=========================================================================*)
6:	(* Scan Fertig *)
	Q_iCnt := 0;
	
	FOR i := 1 TO cMaxScanIDs BY 1 DO 
		IF Q_sIDList[i] <> 0
		THEN
			Q_iCnt := Q_iCnt+1;
		END_IF
	END_FOR
	
	Q_sState := CONCAT('Scan Fertig! Es wurden: ',INT_TO_STRING(Q_iCnt));
	Q_sState := CONCAT(Q_sState,' Teilnehmer gefunden!');
		
	IF rTrigSearch.Q
	THEN
		iStep := 0;
	END_IF
END_CASE

END_FUNCTION_BLOCK

// ---- POUs/RS485_Hausbus_FB/Events/fb_BusPingEvent.TcPOU
FUNCTION_BLOCK fb_BusPingEvent
VAR_INPUT
	 I_sID         			:STRING(10);     // Geräte-ID (z.B. '12345')
	 I_sReceivedString		:STRING(255);	
	 I_bReset				:BOOL;
END_VAR
VAR_OUTPUT
	Q_bOut					:BOOL;
END_VAR
VAR
	findString0				:STRING ;
	findString1				:STRING ;
	findString2				:STRING ;
	findString3				:STRING ;
	findString4				:STRING ;
	findString5				:STRING ;	// Für CYD Ping
END_VAR

(* Wenn ein Taster gedrückt wird *)
findString0 := CONCAT(I_sID,'.');
findString0 := CONCAT(findString0,'BTN');
findString0 := CONCAT(findString0,'.');

(* Wenn ein Relais geschaltet wird *)
findString1 := CONCAT(I_sID,'.');
findString1 := CONCAT(findString1,'OUT');
findString1 := CONCAT(findString1,'.');

(* Wenn Ein Temperatur Event Kommt *)
findString2 := CONCAT(I_sID,'.');
findString2 := CONCAT(findString2,'TMP.1.');

(* Wenn Ein Feuchtigkeit Event Kommt *)
findString3 := CONCAT(I_sID,'.');
findString3 := CONCAT(findString3,'RHD.1.');

(* Wenn Ein Helligkeit Event Kommt *)
findString4 := CONCAT(I_sID,'.');
findString4 := CONCAT(findString4,'BRS.1.');

(* Wenn Ein Display Helligkeits Event Kommt für CYD *)
findString5 := CONCAT(I_sID,'.');
findString5 := CONCAT(findString5,'LBN.16.');

IF I_bReset
THEN
	Q_bOut := FALSE;
ELSE
	IF 	FIND(I_sReceivedString,findString0) >0 
		OR FIND(I_sReceivedString,findString1) >0 
		OR FIND(I_sReceivedString,findString2) >0 
		OR FIND(I_sReceivedString,findString3) >0 
		OR FIND(I_sReceivedString,findString4) >0 
		OR FIND(I_sReceivedString,findString5) >0 
	THEN
		Q_bOut := TRUE;
	ELSE
		Q_bOut := FALSE;
	END_IF
END_IF

END_FUNCTION_BLOCK

// ---- POUs/RS485_Hausbus_FB/BusTaster/fb_TasterBus6F.TcPOU
(*======================================================================================================================================*)
(*FB_TasterBusSimple:	Einfache RS485 Kommunikation für Haus-bus.de Komponenten zum testen 	
						Achtung: Bei dem 6 Fach Taster ist zu Beachten, dass es nur 4 Externe EA/s gibt also 4 LEDs und 4 Taster *)
(*
Date          	| Version    	| created under        	| Author          	| Remark *)
(*====================================================================================================================================================*)
(*29/04/2025   	| 1.00      		| TC3		  		| N.Kersting       | first release *)
(*02/05/2025   	| 1.01      		| TC3		  		| N.Kersting       | Events für die Buttons werden erfolgreich verarbeitet *)
(*02/05/2025   	| 1.02      		| TC3		  		| N.Kersting       | Events für Temp, Helligkeit, Fuehctigkeit erfolgreich Implementier *)
(*02/05/2025   	| 1.03      		| TC3		  		| N.Kersting       | Set Schrittkette für Reset und LED Helligkeit erfolgreich Implementier*)
(*02/05/2025   	| 1.04      		| TC3		  		| N.Kersting       | In und Out Strukturen Implementiert und Startup nach Reset *)
(*02/05/2025   	| 1.05      		| TC3		  		| N.Kersting       | Pingabgfrage*)
(*02/05/2025   	| 1.06      		| TC3		  		| N.Kersting       | Reset Startup Implementiert*)
(*03/05/2025   	| 1.07      		| TC3		  		| N.Kersting       | Ping wird nun bei PLC Reset auch gestaret und Execute wird richtig verwendet*)
(*04/05/2025   	| 1.08      		| TC3		  		| N.Kersting       | Hintergrundbeleuchtung und Zähler für die Tatser Implementiert *)
(*04/05/2025   	| 1.09      		| TC3		  		| N.Kersting       | Neuen Baustein zum Einheitlichen versenden von Telegrammen Implementiert *)
(*05/05/2025   	| 2.00      		| TC3		  		| N.Kersting       | Komplett neuen Baustein, mit Externer Receive Auswertung und neuem Ping Baustein *)
(*06/05/2025   	| 2.01      		| TC3		  		| N.Kersting       | Externe LEDs Implementiert *)
(*07/05/2025   	| 2.02      		| TC3		  		| N.Kersting       | Im Startup wird nun auf die Device ID geachtet *)
(*08/05/2025   	| 2.03      		| TC3		  		| N.Kersting       | Externe LEDs sind nun Umschaltbar/ LEDs oder normaler Ausgang (Betriefft die Hintergrundbeleuchtung) -> Weniger Busauslastung *)
(*09/05/2025   	| 2.04      		| TC3		  		| N.Kersting       | Ping Versuche Implementiert mit Globalen Parametern *)
(*09/05/2025   	| 2.05      		| TC3		  		| N.Kersting       | Ping für Taster nun Auch automatisch durch Empfang von sämtlichen Telegrammen*)
(*09/05/2025   	| 2.06      		| TC3		  		| N.Kersting       | Bugfix im Startup Angepasst! nur noch Hintergrundbeleuchtung setzen! *)
(*10/05/2025   	| 3.00      		| TC3		  		| N.Kersting       | Umstellung auf Externe FiFo Sendebaustein *)
(*13/05/2025   	| 3.01      		| TC3		  		| N.Kersting       | Viele Bugs gefixt, bei Änderung der Ausgängen wird nun eine Anforderung gesetzt  *)
(*13/05/2025   	| 3.02      		| TC3		  		| N.Kersting       | Test für Github *)
(*23/05/2025   	| 3.03      		| TC3		  		| N.Kersting       | Auto - Input Fault Detection implementiert (Wenn Taster zu lange aktiviert bleibt ) *)
(*28/05/2025   	| 3.04      		| TC3		  		| N.Kersting       | Neuen Einfachen Ping Baustein, welcher nicht sendet, nur auswertet implementiert *)
(*====================================================================================================================================================*)
FUNCTION_BLOCK fb_TasterBus6F
VAR_INPUT
	I_FifoID			:INT;
	I_bPingStart		:BOOL;						(* Ping Done vom Vorheriegen*)
	I_stInput			:ST_BusTaster6F_Input;
	I_StringReceived	:STRING(255);
END_VAR
VAR_OUTPUT
	Q_sFiFoSend			:STRING(255);
   	Q_stOutput			:ST_BusTaster6F_Output;
	Q_stCnt				:ST_BusTaster6F_Cnt;
END_VAR
VAR
(*----------------------------------------------*)
(* Interne Parameter*)
(*----------------------------------------------*)		
	bSetExecute			:BOOL := TRUE;				(* Aktiviert die Schrittketten, welche Telegramme versenden *)
	bCheckPing			:BOOL := TRUE;				(* Ping Checken Schrittkette Aktivieren *)
	sStartZeichen		:BYTE := 16#FD;				(* Startzeichen Präfix *)
	sEndZeichen			:BYTE := 16#FE;				(* Endzeichen Suffix *)
	iAnzResetSend		:INT := 2;					(* Anzahl der Sendeversuche bei Reset *)
	tPingTimer			:TIME:= T#5S;				(* Zeit, bis wiederholend der Ping versendet wird *)
	tReceiveTimeout		:TIME:= T#2S;				(* Zeit, bis die Event Schrittkette für das Empfangen Automatisch neu Startet*)
	tStartupLEDOn		:TIME:= T#4S;				(* Zeit, wie Lange die LEDS beim Startup kurz eingeschaltet werden *)
	tResetTimeout		:TIME:= T#10S;				(* Zeit, bis bei einem Reset es zu einem Fehler kommt, wenn kein Ping empfangen wird *)
	tResetReboot		:TIME:= T#10S;				(* Zeit, die nach einem Reset Abgewaretet wird damit das Gerät neustarten kann*)
	tResetStartup		:TIME:= T#5S;				(* Zeit, die nach einem Reset Abgewaretet wird bis ein Startup ausgeführt wird nach dem erhalt des Pings vom Gerät*)
	tStartupAfterReset	:TIME := T#5S;				(* Zeit, wann das Startup Zurückgesetzt wird, wenn der Ping verloren wird *)
	bInputFaultDetect	:BOOL := TRUE;				(* Prüft die Eingänge ob sie zu lange geschaltet wurden und führt ein reset des eingangs aus *)
	tInputFaultDetect	:TIME := T#10S;				(* Prüft die Eingänge ob sie zu lange geschaltet wurden und führt ein reset des eingangs aus *)
(*----------------------------------------------*)
(* Strings *)
(*----------------------------------------------*)			
	sSendString			:STRING(255);
	sFiFoSend			:STRING(255);
	sReceived			:STRING(255);
	sLastSendString		:STRING(255);
	sStateReset			:STRING;
(*----------------------------------------------*)
(* Funktionsbausteine *)
(*----------------------------------------------*)
	fbBusTasterEvent	:ARRAY[1..6] OF fb_BusTasterEvent;		(* Interne 6 Taster Abfragen *)
	fbBusTasterEventExt	:ARRAY[1..6] OF fb_BusTasterEvent;		(* Externe 6 Eingänge Abfragen *)
	fbBusTempEvent		:fb_BusTempEvent;
	fbBusBrsEvent		:fb_BusBrsEvent;
	fbBusRhdEvent		:fb_BusRhdEvent;
	fbStringConvTB6F	:fb_StringConvTB6F;
	fbPing				:fb_RS485Ping;
(*----------------------------------------------*)
(* Indexe *)
(*----------------------------------------------*)	
	iDeviceStartup		:INT :=0;	(* Startup Schrittkette *)
	sDeviceStartup		:STRING;
    iState     			:INT := 0;
	iStepSet			:INT;
	i,h,j,l,e			:INT;
	idxLED				:INT;
	idxBtn				:INT := 1;
	
	iDimmMem			:ARRAY[1..6] OF INT;
	iDimmMemExt			:ARRAY[1..6] OF INT;
	iDimmBGAnf			:INT;
	iDimmAnf			:ARRAY[1..6] OF INT;
	iDimmAnfExt			:ARRAY[1..6] OF INT;
	
	iDimmBgMem			:INT;
	cntChangesDimm		:INT;
	cntChangesDimmExt	:INT;
	icntResetSend		:INT;
	iMaxPingTry			:INT := 5;
(*----------------------------------------------*)
(* Timer/Trigger *)
(*----------------------------------------------*)		
	r_trigStartupAfterReset	:r_trig;
	r_TrigReset				:r_trig;		
	r_TrigCountBtn			:ARRAY[1..6] OF r_trig;
	
	tonStartupAfterReset	:ton;
	tonReceiveTimeout		:ton;
	tonResetTimeout			:ton;
	tonResetDone			:ton;
	tonStepStartup			:ton;
(*----------------------------------------------*)
(* Status *)
(*----------------------------------------------*)			
	bPingOK					:BOOL;
	bErrorEvent				:BOOL;
	bErrorPing				:BOOL;
	bErrorSet				:BOOL;
	bErrorReset				:BOOL;
	bResetBusy				:BOOL;
	bResetDone				:BOOL;
	bResetAutoStart			:BOOL;
	bStartupStart			:BOOL;
	bStartupDone			:BOOL;	
	bMemExt					:BOOL;
	bStartUpCheckPing		:BOOL;
	bActivateSend			:BOOL;
	bReadyToPing			:BOOL;
	bSendeAnforderung		:BOOL;
	bSendeAnforderungExt	:BOOL;
	bSendeAnforderungBG		:BOOL;
	
END_VAR

(*============================================================================================*)
(* Parameter *)
tPingTimer :=		GVL_HausBus_Parameter.cTimePingTimeTaster;
tReceiveTimeout :=	GVL_HausBus_Parameter.cTimeReceiveTimeoutTaster;
bCheckPing :=		GVL_HausBus_Parameter.bUseTasterPing;
iMaxPingTry :=		GVL_HausBus_Parameter.cMaxPingTry;

(*============================================================================================*)
(* Startup Zurücksetzen Reset *)
r_TrigReset(CLK := I_stInput.bReset);

(* Startup Zurücksetzen bei Busverlust *)
tonStartupAfterReset(
	IN := NOT bPingOK
			AND bCheckPing,
	PT:= tStartupAfterReset);

r_trigStartupAfterReset
	(CLK := tonStartupAfterReset.Q);
	
IF NOT I_stInput.bExecute
	OR r_TrigReset.Q
	OR r_trigStartupAfterReset.Q
THEN
	iDeviceStartup := 0;
END_IF

(*============================================================================================*)
(* Ping Dauerhaft Senden*)
ac02_Ping();
	
(*============================================================================================*)
(* Startup Schrittkette *)
CASE iDeviceStartup OF
(*============================================================================================*)
0: 	sDeviceStartup := 'INIT';
	bResetDone := FALSE;
	bStartupDone := FALSE;
	bStartupStart := FALSE;
	bResetAutoStart := FALSE;
	bStartUpCheckPing := FALSE;
	bActivateSend := FALSE;
	bReadyToPing := TRUE;
	sFiFoSend := ''; 
	iStepSet := 0;
	
	IF 	I_stInput.bExecute
	THEN
		iDeviceStartup := iDeviceStartup+1;
	END_IF
(*============================================================================================*)
1: 	sDeviceStartup := 'Device ID Prüfen';
	
	IF  I_stInput.diID <> 0
	THEN
		iDeviceStartup := iDeviceStartup+1;
	ELSE
		sDeviceStartup := 'ERROR- Device ID Prüfen';
	END_IF
(*============================================================================================*)
2: 	sDeviceStartup := 'Verbindung Prüfen';
	bActivateSend := TRUE;	(* Senden Aktivieren *)
	iDeviceStartup := iDeviceStartup+1;
	
	(*
	sDeviceStartup := CONCAT(sDeviceStartup,fbRS485ComCheck.Q_sState);
	
	IF fbRS485ComCheck.Q_bComOk
		OR NOT bCheckPing
	THEN
		iDeviceStartup := iDeviceStartup+1;
	END_IF*)

(*============================================================================================*)
3: 	sDeviceStartup := 'Reset Ausführen';	
	bActivateSend := TRUE;	(* Senden Aktivieren *)
	
	(*	RESET Device *)
	ac01_SetReset();
	bResetAutoStart := TRUE;
	
	sDeviceStartup :=	CONCAT(sDeviceStartup,sStateReset);
	
	IF bResetDone
	THEN
		iStepSet := 0;
		iDeviceStartup := iDeviceStartup+1;
	END_IF

(*============================================================================================*)
4: 	sDeviceStartup := 'Startup Ausführen';
		
	(* LED Setzen *)
	ac01_SetLED();
	
	bStartupStart := TRUE;
	
	IF bStartupDone 
	THEN
		bStartupStart := FALSE;
		iDeviceStartup := 999;
	END_IF

(*============================================================================================*)
999: 
	(*bReadyToPing := NOT fbRS485SendCmd.Q_bBusy;*)
		
	(* LED Setzen *)
	ac01_SetLED();
	
	(* Events Auslesen *)
	ac00_Event();
	
	(* Zähler *)
	ac10_Counter();
	
	sDeviceStartup := 'Startup Ausgeführt- Gerät im OP';
	
END_CASE

(*============================================================================================*)
(* Sendebaustein *)
IF bActivateSend
THEN
	Q_sFiFoSend :=	sFiFoSend;
END_IF

(*============================================================================================*)	
(* Zähler *)
ac10_Counter();
	
(*============================================================================================*)
(* Outputs *)
Q_stOutput.bCOM :=		bPingOK;

Q_stOutput.bError := 	bErrorEvent
						OR bErrorPing
						OR bErrorSet
						OR (NOT bPingOK
						AND bCheckPing);
						
Q_stOutput.bStartupDone	:=	bStartupDone;

Q_stOutput.sState :=	CONCAT(I_stInput.sName,'| ');
Q_stOutput.sState :=	CONCAT(Q_stOutput.sState, sDeviceStartup);

ACTION ac00_Event:
(*============================================================================================*)
(*	EVENT Schrittkette *)
(*============================================================================================*)
sReceived := I_StringReceived;
	
FOR i := 1 TO 6 BY 1 DO 
	
	fbBusTasterEvent[i](
		I_bFaultDetection	:=	bInputFaultDetect,
		I_tFaultDetectTime	:=	tInputFaultDetect,
		I_sID:= 				DINT_TO_STRING(I_stInput.diID), 
		I_sInstID:= 			INT_TO_STRING(i+16), 
		I_sReceivedString:= 	sReceived, 
		Q_bOut=> 				Q_stOutput.bButtons[i]);
	
	fbBusTasterEventExt[i](
		I_sID:= 				DINT_TO_STRING(I_stInput.diID), 
		I_sInstID:= 			INT_TO_STRING(i+32), 
		I_sReceivedString:= 	sReceived, 
		Q_bOut=> 				Q_stOutput.bButtonsExt[i]);
		
	fbBusTempEvent(
		I_sID:= 				DINT_TO_STRING(I_stInput.diID), 
		I_sInstID:= 			'1', 
		I_sReceivedString:= 	sReceived, 
		Q_lrTemp=> 				Q_stOutput.lrTemp);
		
	fbBusBrsEvent(
		I_sID:= 				DINT_TO_STRING(I_stInput.diID), 
		I_sInstID:= 			'1', 
		I_sReceivedString:= 	sReceived, 
		Q_lrBrs=> 				Q_stOutput.lrBrs);
		
	fbBusRhdEvent(
		I_sID:= 				DINT_TO_STRING(I_stInput.diID), 
		I_sInstID:= 			'1', 
		I_sReceivedString:= 	sReceived, 
		Q_lrRhd=> 				Q_stOutput.lrRhd);
END_FOR
END_ACTION

ACTION ac01_SetLED:
(*============================================================================================*)
(*	LED Helligkeit Setzen/ Startup Schrittkette *)
(*============================================================================================*)

(* Einfaches Setzen der LED Helligkeiten (0-100 Prozent *)
(* Neu, es werden alle LEDs zu einem String zusammengefügt und Gleichzeitig gesetzt *)
tonStepStartup(
	PT:= tStartupLEDOn);
	
cntchangesDimm := 0;
cntChangesDimmExt :=0;
	
FOR l := 1 TO 6 BY 1 DO
	IF iDimmMem[l] <> I_stInput.iLED[l]
	THEN
		cntChangesDimm := cntChangesDimm +1;
	END_IF

	IF  iDimmMemExt[l]<> I_stInput.iLEDExt[l]
	THEN
		cntChangesDimmExt := cntChangesDimmExt +1;
	END_IF
END_FOR

CASE iStepSet OF
(*============================================================================================*)
0:	(* INIT und warten auf Change *)				
	tonStepStartup.IN := FALSE;
	sFiFoSend := ''; 
	
	(* Änderungs- Anforderungen Prüfen*)
	FOR e := 1 TO 6 BY 1 DO
		IF cntChangesDimm<>0
		THEN
			(* Helligkeitanforderung Interne LEDs speichern *)
			bSendeAnforderung := TRUE;
			iDimmAnf[e] 	:= I_stInput.iLED[e];
		END_IF
		
		IF cntChangesDimmExt <> 0
		THEN
			(* Helligkeitanforderung Externe LEDs speichern *)
			bSendeAnforderungExt := TRUE;
			iDimmAnfExt[e] 	:= I_stInput.iLEDExt[e];
		END_IF
		
		IF I_stInput.iLEDBg <>iDimmBgMem
		THEN
			(* Helligkeitsanforderung Hintergrundbeleuchtung *)
			bSendeAnforderungBG := TRUE;
			iDimmBGAnf		:= I_stInput.iLEDBg;
		END_IF
	END_FOR
	
	(* Reagieren auf Anforderungen *)
	IF ((bSendeAnforderung
		OR bSendeAnforderungExt
		OR bSendeAnforderungBG)
		AND bSetExecute)
		AND NOT bStartupStart
	THEN
		(* Helligkeitsvorgaben speichern in Mem Arrays *)
		FOR h := 1 TO 6 BY 1 DO
			iDimmMem[h] := I_stInput.iLED[h];
			iDimmMemExt[h] := I_stInput.iLEDExt[h];
			iDimmBgMem := I_stInput.iLEDBg;
		END_FOR
		
		iStepSet := 10;
	ELSIF
		bStartupStart
	THEN
		iStepSet := 100;	(* Startup *)
	END_IF
	
(*============================================================================================*)
10:	(* Prüfen welche Anforderung ausgeführt werden soll *)	
	IF	bSendeAnforderungBG
		AND NOT bSendeAnforderung
		AND NOT bSendeAnforderungExt 
	THEN
		iStepSet := 22;(* Direkt nur die Hintergrund Helligkeit setzen *)
	ELSE
		(* Nur Interne LEDs Schreiben *)
		IF bSendeAnforderung
			AND NOT bSendeAnforderungExt
			AND NOT bSendeAnforderungBG
		THEN
			fbStringConvTB6F(
				I_bSetBackground :=	FALSE,
				I_bReset :=			FALSE,
				I_bExtLED :=		FALSE,
				I_bHasExtLED :=		I_stInput.bExtOutLED,
				I_diID:= 			I_stInput.diID, 
				I_iLED:= 			iDimmAnf, 
				I_iLEDExt:=			iDimmAnfExt,
				I_iLEDBg:= 			iDimmBGAnf,		 
				I_sStartZeichen:= 	sStartZeichen, 
				I_sEndZeichen:= 	sEndZeichen, 
				Q_sConvString=> 	sSendString);
				
			(* Senden an FiFo*)
			IF GVL_RS485FiFoSend.bSendDoneFiFo[I_FifoID]
			THEN
				sFiFoSend :=	sSendString;
			END_IF
			IF NOT GVL_RS485FiFoSend.bSendDoneFiFo[I_FifoID]
			THEN
				bSendeAnforderung := FALSE;
				sLastSendString :=	sFiFoSend;
				iStepSet := 20;
			END_IF
		ELSIF
			(* Nur Externe LEDs Schreiben *)	
			bSendeAnforderungExt
			AND NOT bSendeAnforderung
			AND NOT bSendeAnforderungBG
		THEN
			fbStringConvTB6F(
				I_bSetBackground :=	FALSE,
				I_bReset :=			FALSE,
				I_bExtLED :=		TRUE,
				I_bHasExtLED :=		I_stInput.bExtOutLED,
				I_diID:= 			I_stInput.diID, 
				I_iLED:= 			iDimmAnf, 
				I_iLEDExt:=			iDimmAnfExt,
				I_iLEDBg:= 			iDimmBGAnf,				 
				I_sStartZeichen:= 	sStartZeichen, 
				I_sEndZeichen:= 	sEndZeichen, 
				Q_sConvString=> 	sSendString);
			
			(* Senden an FiFo*)
			IF GVL_RS485FiFoSend.bSendDoneFiFo[I_FifoID]
			THEN
				sFiFoSend :=	sSendString;
			END_IF
			IF NOT GVL_RS485FiFoSend.bSendDoneFiFo[I_FifoID]
			THEN
				bSendeAnforderungExt := FALSE;
				sLastSendString :=	sFiFoSend;
				iStepSet := 20;
			END_IF
		ELSE
			(* Externe und Interne LEDs Schreiben *)
			bMemExt := TRUE; (* Speichern, damit anschließend noch die Externen LEDs gesetzt werden *)
			
			fbStringConvTB6F(
				I_bSetBackground :=	FALSE,
				I_bReset :=			FALSE,
				I_bExtLED :=		FALSE,
				I_bHasExtLED :=		I_stInput.bExtOutLED,
				I_diID:= 			I_stInput.diID, 
				I_iLED:= 			iDimmAnf, 
				I_iLEDExt:=			iDimmAnfExt,
				I_iLEDBg:= 			iDimmBGAnf,			 
				I_sStartZeichen:= 	sStartZeichen, 
				I_sEndZeichen:= 	sEndZeichen, 
				Q_sConvString=> 	sSendString);
			
			(* Senden an FiFo*)
			IF GVL_RS485FiFoSend.bSendDoneFiFo[I_FifoID]
			THEN
				sFiFoSend :=	sSendString;
			END_IF
			IF NOT GVL_RS485FiFoSend.bSendDoneFiFo[I_FifoID]
			THEN
				bSendeAnforderung := FALSE;
				bSendeAnforderungExt := FALSE;
				sLastSendString :=	sFiFoSend;
				iStepSet := 20;
			END_IF
		END_IF
	END_IF
(*============================================================================================*)	
20:	(* Warten bis nicht Busy *)	
	
	IF GVL_RS485FiFoSend.bSendDoneFiFo[I_FifoID]
	THEN
		sFiFoSend := ''; 
		IF NOT bMemExt
		THEN
			IF bSendeAnforderungBG
			THEN
				iStepSet := 22;
			ELSE
				iStepSet := 0;
			END_IF
		ELSE
			iStepSet :=	21;
		END_IF
	END_IF
	
(*============================================================================================*)	
21:	(* Externe LEDs Senden *)	
	bMemExt := FALSE;
	bSendeAnforderungExt := FALSE;
	
	fbStringConvTB6F(
		I_bSetBackground :=	FALSE,
		I_bReset :=			FALSE,
		I_bExtLED :=		TRUE,
		I_bHasExtLED :=		I_stInput.bExtOutLED,
		I_diID:= 			I_stInput.diID, 
		I_iLED:= 			iDimmAnf, 
		I_iLEDExt:=			iDimmAnfExt,
		I_iLEDBg:= 			iDimmBGAnf,				 
		I_sStartZeichen:= 	sStartZeichen, 
		I_sEndZeichen:= 	sEndZeichen, 
		Q_sConvString=> 	sSendString);
		
	(* Senden an FiFo*)
	IF GVL_RS485FiFoSend.bSendDoneFiFo[I_FifoID]
	THEN
		sFiFoSend :=	sSendString;
	END_IF
	IF NOT GVL_RS485FiFoSend.bSendDoneFiFo[I_FifoID]
	THEN
		sLastSendString :=	sFiFoSend;
		iStepSet := 20;
	END_IF
	
(*============================================================================================*)	
22:	(* Hintergrundbeleuchtung senden *)		
	bSendeAnforderungBG := FALSE;
	
	fbStringConvTB6F(
		I_bSetBackground :=	TRUE,
		I_bReset :=			FALSE,
		I_bExtLED :=		FALSE,
		I_bHasExtLED :=		I_stInput.bExtOutLED,
		I_diID:= 			I_stInput.diID, 
		I_iLED:= 			iDimmAnf, 
		I_iLEDExt:=			iDimmAnfExt,
		I_iLEDBg:= 			iDimmBGAnf,			 
		I_sStartZeichen:= 	sStartZeichen, 
		I_sEndZeichen:= 	sEndZeichen, 
		Q_sConvString=> 	sSendString);
		
	(* Senden an FiFo*)
	IF GVL_RS485FiFoSend.bSendDoneFiFo[I_FifoID]
	THEN
		sFiFoSend :=	sSendString;
	END_IF
	IF NOT GVL_RS485FiFoSend.bSendDoneFiFo[I_FifoID]
	THEN
		sLastSendString :=	sFiFoSend;
		iStepSet := 20;
	END_IF

(*============================================================================================*)	
(* Startup LEDS einmal Einschalten *)
100:	tonStepStartup.IN := TRUE;
	
	IF tonStepStartup.Q
	THEN
		iStepSet := 110;
	END_IF
	
(*============================================================================================*)
110:	(* String senden *)	
	tonStepStartup.IN := FALSE;
	
	fbStringConvTB6F(
		I_bSetBackground :=	TRUE,
		I_bExtLED :=		FALSE,
		I_bReset :=			FALSE,
		I_bHasExtLED :=		I_stInput.bExtOutLED,
		I_diID:= 			I_stInput.diID, 
		I_iLEDBg:= 			100,		 
		I_sStartZeichen:= 	sStartZeichen, 
		I_sEndZeichen:= 	sEndZeichen, 
		Q_sConvString=> 	sSendString);
			
	(* Senden an FiFo*)
	IF GVL_RS485FiFoSend.bSendDoneFiFo[I_FifoID]
	THEN
		sFiFoSend :=	sSendString;
	END_IF
	IF NOT GVL_RS485FiFoSend.bSendDoneFiFo[I_FifoID]
	THEN
		
		iStepSet := 111;
	END_IF
	
(*============================================================================================*)	
111:(* Warten bis nicht Busy *)	
	IF GVL_RS485FiFoSend.bSendDoneFiFo[I_FifoID]
	THEN
		sFiFoSend := ''; 
		tonStepStartup.IN := TRUE;
		
		IF tonStepStartup.Q
		THEN
			tonStepStartup.IN := FALSE;
			iStepSet := 120;
		END_IF
	END_IF
	
(*============================================================================================*)
120:	(* String senden *)	
	fbStringConvTB6F(
		I_bSetBackground :=	TRUE,
		I_bExtLED :=		FALSE,
		I_bReset :=			FALSE,
		I_bHasExtLED :=		I_stInput.bExtOutLED,
		I_diID:= 			I_stInput.diID, 
		I_iLEDBg:= 			0,		 
		I_sStartZeichen:= 	sStartZeichen, 
		I_sEndZeichen:= 	sEndZeichen, 
		Q_sConvString=> 	sSendString);
			
	(* Senden an FiFo*)
	IF GVL_RS485FiFoSend.bSendDoneFiFo[I_FifoID]
	THEN
		sFiFoSend :=	sSendString;
	END_IF
	IF NOT GVL_RS485FiFoSend.bSendDoneFiFo[I_FifoID]
	THEN
		iStepSet := 130;
	END_IF
	
(*============================================================================================*)	
130:(* Warten bis nicht Busy *)	
	IF GVL_RS485FiFoSend.bSendDoneFiFo[I_FifoID]
	THEN
		sFiFoSend := ''; 
			
		tonStepStartup.IN := TRUE;
	
		IF tonStepStartup.Q
		THEN
			bStartupDone := TRUE;
			tonStepStartup.IN := FALSE;
			bStartupStart := FALSE;
			iStepSet := 10;	(* Anschließend noch einmal die Eingangs Helligkeit setzen *)
		END_IF
	END_IF	

END_CASE

(*bErrorSet := fbRS485SendCmd.Q_bError;*)
END_ACTION

ACTION ac01_SetReset:
(*============================================================================================*)
(*	RESET Schrittkette *)
(*============================================================================================*)
tonResetTimeout(
	PT := tResetTimeout);

tonResetDone();

(* Einfaches Setzen der LED Helligkeiten (0-100 Prozent *)
CASE iStepSet OF
(*============================================================================================*)
0:	sStateReset := 'INIT';
	
	IF (bSetExecute
		AND (I_stInput.bReset
		OR bResetAutoStart))
	THEN
		sFiFoSend := ''; 
		bStartupDone := FALSE;
		bResetDone := FALSE;
		tonResetTimeout.IN := FALSE;
		tonResetDone.IN := FALSE;
		icntResetSend := 0;
		
		(* Ausgänge alle auf 0 setzen *)
		FOR h := 1 TO 6 BY 1 DO
			fbBusTasterEvent[i](
				I_sReceivedString :='');
				
			fbBusTasterEventExt[i](
				I_sReceivedString :='');	
				
			iDimmMem[h] := 0;
			Q_stOutput.bButtons[h] := FALSE;
			Q_stOutput.lrTemp := 0;
			Q_stOutput.lrBrs := 0;
			Q_stOutput.lrRhd := 0;
		END_FOR
		
		fbBusTempEvent(
			I_sReceivedString :='',	
			I_bReset := TRUE);
			
		fbBusBrsEvent(
			I_sReceivedString :='',	
			I_bReset := TRUE);
			
		fbBusRhdEvent(
			I_sReceivedString :='',	
			I_bReset := TRUE);
		
		bPingOK := FALSE;
		
		iStepSet := iStepSet +1;
	END_IF

(*============================================================================================*)	
1:	sStateReset := 'Sende Reset Befehl';
	bResetBusy := TRUE;
	bErrorReset := FALSE;
	
	fbStringConvTB6F(
		I_bReset :=			TRUE,
		I_diID:= 			I_stInput.diID, 		 
		I_sStartZeichen:= 	sStartZeichen, 
		I_sEndZeichen:= 	sEndZeichen, 
		Q_sConvString=> 	sSendString);

	(* Senden an FiFo*)
	IF GVL_RS485FiFoSend.bSendDoneFiFo[I_FifoID]
	THEN
		sFiFoSend :=	sSendString;
	END_IF
	IF NOT GVL_RS485FiFoSend.bSendDoneFiFo[I_FifoID]
	THEN
		iStepSet := iStepSet+1;
	END_IF

(*============================================================================================*)
2:	sStateReset := 'Sende Reset Befehl';

	IF GVL_RS485FiFoSend.bSendDoneFiFo[I_FifoID]
	THEN
		sFiFoSend := ''; 
		fbStringConvTB6F(
			I_bReset :=			FALSE);
		iStepSet := 3;
				
	END_IF
	
(*============================================================================================*)	
3:	sStateReset := 'Reset durchgeführt, Warte auf Ping';
	tonResetDone.IN := TRUE;
	tonResetDone.PT := tResetReboot;
	
	fbBusTempEvent(I_bReset := FALSE);
	fbBusBrsEvent(I_bReset := FALSE);
	fbBusRhdEvent(I_bReset := FALSE);
	
	iState := 0;
	
	IF tonResetDone.Q
	THEN
		tonResetDone.IN := FALSE;
		iStepSet := 4;
	END_IF
	
(*============================================================================================*)	
4:	sStateReset := 'Warte auf Ping vom Gerät';	
	tonResetTimeout.IN := TRUE;
	bStartUpCheckPing := TRUE;
	
	IF bPingOK 
		(*OR NOT bCheckPing*)
	THEN
		bErrorReset := FALSE;
		tonResetTimeout.IN := FALSE;
		iStepSet := 5;
	ELSIF
		tonResetTimeout.Q
	THEN
		sStateReset := 'Ping Timeout, keine Kommunikation';
		bErrorReset := TRUE;

		IF I_stInput.bReset
		THEN
			bResetBusy := FALSE;
			iStepSet := 0;
		END_IF
	END_IF

(*============================================================================================*)
5:	sStateReset := 'Startup Aktiv';
	
	tonResetDone.IN := NOT I_stInput.bReset;
	tonResetDone.PT := tResetStartup;
	sFiFoSend := ''; 
	
	IF tonResetDone.Q
	THEN
		fbStringConvTB6F(
			I_bReset :=			FALSE);
			
		sStateReset := 'Ping erhalten, Reset Erfolgreich';
		bResetAutoStart := FALSE;
		bResetDone := TRUE;
		bResetBusy := FALSE;
		iState := 0;
		iStepSet := 0;
	END_IF
END_CASE
END_ACTION

ACTION ac02_Ping:
(*============================================================================================*)
(* 	Ping Bautsein, Checkt ob die Kommunikation vorhanden ist *)
(*============================================================================================*)
fbPing(
	I_bExecute:= 			bStartUpCheckPing, 
	I_bAutoPing:= 			bCheckPing, 
	I_bAutoReset:= 			bCheckPing, 
	I_bReset:= 				r_TrigReset.Q
							OR NOT bStartUpCheckPing, 
	I_tPingTimeout:= 		tPingTimer, 
	I_diID:= 				I_stInput.diID, 
	I_sStartZeichen:= 		sStartZeichen, 
	I_sEndZeichen:= 		sEndZeichen, 
	I_StringReceived:= 		I_StringReceived, 
	Q_sState=> , 
	Q_bComOk=> 				bPingOK, 
	Q_bTimeout=> 			bErrorPing);
END_ACTION

ACTION ac10_Counter:
(*============================================================================================*)
(* 	Zähler *)
(*============================================================================================*)
FOR j := 1 TO 6 BY 1 DO 
	r_TrigCountBtn[j](
		CLK := Q_stOutput.bButtons[j]);
		
	IF r_TrigCountBtn[j].Q
	THEN
		Q_stCnt.dwCntButtons[j] := Q_stCnt.dwCntButtons[j]+1;
	END_IF
	
END_FOR
END_ACTION

ACTION ac99_Doku:
(*======================================================================================================================================*)
(*	DOKU	*)
(*======================================================================================================================================*)
(* Wichtiger Hinweis:
		-Bei dem 6 Fach Taster ist zu Beachten, dass es nur 4 Externe EA/s gibt also 4 LEDs und 4 Taster, 
		da der ESP 32 Nur 10Es und 10As besitzt.
		- Die 4 Zusätzlichen Ausgänge werden von der Hintergrundbeleuchtung Ausgeschlossen und müssen über den Befehl: SET_MBR einzeln 
			gesetzt werden! *)	
	
(* Verdrahtung:		
	Verdrahtung füR: KL6041
        +-------+
        |       |
        | TxD+ ----+
        |         |----> RS485 A (zum Bus)
        | RxD+ ----+
        |         |
        | TxD− ----+
        |         |----> RS485 B (zum Bus)
        | RxD− ----+
        +-------+	*)
		
(*======================================================================================================================================*)
(* Telegrammbeschreibung *)

(*	Die XML Dateien der verschiedenen Module sind grundsätzlich immer gleich aufgebaut. 
	Je Instanz der verschiedenen Sensoren und Aktoren werden die zu sendenden Befehle bzw. 
	die zu empfangenen Events beschrieben. 
	Alle Telegramme sind ASCII kodiert und sind umgeben mit dem binären Startzeichen 0xFD und dem binären Endezeichen 0xFE.

	Grundaufbauer aller im Folgenden beschriebenen Telegramme:
	
	-Startzeichen immer 0xFD.
	-Punkte dienen als Trennzeichen der verschiedenen Elemente
	-Endezeichen immer 0xFE.
	-Element 1 ist die Geräte-ID, die entsprechend der verwendeten Module angepasst werden muss (hier beispielhaft jeweils 12345)
	-Element 2 ist ein Schlüsselwort für den jeweiligen Funktionstyp (z.b. BTN, LED, DIM, usw)
	-Element 3 ist die InstanzID gemäß XML Templates (also welche Taster oder welcher Dimmer konkret gemeint ist)
	-Element 4 zeigt die jeweilige Aktion zum Funktionstypen (z.b. ON, OFF, STATUS)
	-Anschließend kommen optional diverse Parameter, die mit P1,P2,...P3 bezeichnet werden
	
	Im Folgenden wird nur noch auf die speziellen Telegramdaten eingegangen:
	
	(*------------------------------------------------------------*)
	Taster oder digitaler Eingang (Sensor):
	(*------------------------------------------------------------*)
	Telegram Event:  	
	
	\xFD 12345.BTN.17.STATUS.P1 \xFE
	
		Funktionstyp:		BTN (kurz für Button)
		Instanz-ID:			hier 17 (in XML nachschauen)
		Aktion:				STATUS
		P1:					1, wenn Taste gedrückt bzw. Eingang aktiv
							0, wenn Taste losgelassen bzw. Eingang inaktiv
	
	Telegram Statusabfrage:  	
	
	\xFD 12345.BTN.17.gSTATUS \xFE
	
		Antwort:  			\xFD 12345.BTN.17.rSTATUS.P1 \xFE
		P1:					1, wenn Taste gedrückt bzw. Eingang aktiv
							0, wenn Taste losgelassen bzw. Eingang inaktiv

	(*------------------------------------------------------------*)
	Led (Aktor):
	(*------------------------------------------------------------*)
	Telegram Helligkeit setzen:  	
	
	\xFD 12345.LED.50.ON.P1.P2.P3 \xFE
	
		Funktionstyp:			LED
		Instanz-ID:				hier 50 (in XML nachschauen)
		Aktion:					ON
		P1:						gewünschte Helligkeit 0-100
		P2:						Einschaltdauer in 100stel Sekunden (0 = daueran)
		P3:						Einschaltverzögerung in Sekunden (0 = ohne Verzögerung)
	
	Telegram Mindesthelligkeit:  	
	
	\xFD 12345.LED.50.SET_MBR.P1 \xFE
		
		Aktion:					SET_MBR (Setzt eine Mindesthelligkeit, die auch dann erhalten bleibt, wenn man per OFF ausschaltet)
		P1:						gewünschte Helligkeit 0-100
	
	Telegram Statusabfrage:  	

	\xFD 12345.LED.50.gSTATUS \xFE
	
		Antwort:  				\xFD 12345.LED.50.rSTATUS.P1.P2 \xFE
		P1:						aktuelle Helligkeit 0-100
		P2:						Einschaltdauer in 100stel Sekunden
	
	(*------------------------------------------------------------*)
	Hintergrundbeleuchtung (Aktor):
	(*------------------------------------------------------------*)
	Telegram Minhelligkeit:  
	
	\xFD 12345.LBN.16.SET_MBR.P1 \xFE
	
		Aktion:					SET_MBR ((Setzt eine Mindesthelligkeit, die auch dann erhalten bleibt, wenn man per OFF ausschaltet)
		P1:						gewünschte Helligkeit 0-100
		
	Telegram Statusabfrage:  	

	\xFD 12345.LBN.16.gSTATUS \xFE
	
		Antwort:  				\xFD 12345.LBN.16.rSTATUS.P1 \xFE
		P1:						aktuelle Helligkeit 0-100

	(*------------------------------------------------------------*)
	Temperatursensor (Sensor):
	(*------------------------------------------------------------*)
	Telegram Event:  	
	
	\xFD 12345.TMP.1.STATUS.P1.P2 \xFE
	
		Funktionstyp:			TMP (kurz für Temperatur)
		Instanz-ID:				hier 1 (in XML nachschauen)
		Aktion:					STATUS
		P1:						Temperatur in Grad Vorkommastellen
		P2:						Temperatur in Grad Nachkommastellen
	
	Telegram Statusabfrage:  
	
	\xFD 12345.TMP.1.gSTATUS \xFE
	
		Antwort:  				\xFD 12345.TMP.1.rSTATUS.P1.P2 \xFE
		P1:						Temperatur in Grad Vorkommastellen
		P2:						Temperatur in Grad Nachkommastellen

	(*------------------------------------------------------------*)
	Feuchtesensor (Sensor):
	(*------------------------------------------------------------*)
	Telegram Event:  	

	\xFD 12345.RHD.1.STATUS.P1.P2 \xFE
	
		Funktionstyp:			RHD (kurz für Relative Humidity)
		Instanz-ID:				hier 1 (in XML nachschauen)
		Aktion:					STATUS
		P1:						Relative Luftfeuchtigkeit 0-100 Vorkommastellen
		P2:						Relative Luftfeuchtigkeit 0-100 Nachkommastellen

	Telegram Statusabfrage:  	
	
	\xFD 12345.RHD.1.gSTATUS \xFE
	
	Antwort:  					\xFD 12345.RHD.1.rSTATUS.P1 \xFE
	P1:							Relative Luftfeuchtigkeit 0-100 Vorkommastellen
	P2:							Relative Luftfeuchtigkeit 0-100 Nachkommastellen

	(*------------------------------------------------------------*)
	Helligkeitssensor (Sensor):
	(*------------------------------------------------------------*)
	Telegram Event:  	
	
	\xFD 12345.BRS.23.STATUS.P1.P2 \xFE
	
		Funktionstyp:			BRS (kurz für Brightness Sensor)
		Instanz-ID:				hier 23 (in XML nachschauen)
		Aktion:					STATUS
		P1:						Relative Helligkeit 0-255 Vorkommastellen
		P2:						Relative Helligkeit 0-255 Nachkommastellen
	
	Telegram Statusabfrage:  	
	
	\xFD 12345.BRS.23.gSTATUS \xFE
	
	Antwort:  					\xFD 12345.BRS.23.rSTATUS.P1 \xFE
	P1:							Relative Helligkeit 0-255 Vorkommastellen
	P2:							Relative Helligkeit 0-255 Nachkommastellen

(*======================================================================================================================================*)
(* Alle Telegramme im Überblick *)	

	<?xml version="1.0" encoding="utf-8"?>
	<Comm Title="Haus-Bus ID 12345" Comment="" Baudrate="57600" Databits="8" Parity="1" EndChar="510">
	<CommCmd Title="6-fach Taster 12345 - Hintergrundbeleuchtung" Comment="" CmdOn="\xFD12345.LBN.16.SET_MBR.&lt;v&gt;.0\xFE" CmdOff="\xFD12345.LBN.16.SET_MBR.0\xFE" Unit="" Analog="true" Text="false" Sensor="false" SourceValHigh="100" DestValHigh="100"/>
	<CommCmd Title="6-fach Taster 12345 - Temperatursensor" Comment="" CmdOn="\xFD12345.TMP.1.STATUS.\v\xFE" CmdOff="" Unit="&lt;v.2&gt;" Analog="true" Text="false" Sensor="true" SourceValHigh="100" DestValHigh="100"/>
	<CommCmd Title="6-fach Taster 12345 - Feuchtesensor" Comment="" CmdOn="\xFD12345.RHD.1.STATUS.\v\xFE" CmdOff="" Unit="&lt;v.x&gt;" Analog="true" Text="false" Sensor="true" SourceValHigh="100" DestValHigh="100"/>
	<CommCmd Title="6-fach Taster 12345 - Helligkeitssensor" Comment="" CmdOn="\xFD12345.BRS.1.STATUS.\v\xFE" CmdOff="" Unit="&lt;v.x&gt;" Analog="true" Text="false" Sensor="true" SourceValHigh="100" DestValHigh="100"/>
	<CommCmd Title="6-fach Taster 12345 - Led 1" Comment="" CmdOn="\xFD12345.LED.49.ON.&lt;v&gt;.0\xFE" CmdOff="\xFD12345.LED.49.OFF\xFE" Unit="" Analog="true" Text="false" Sensor="false" SourceValHigh="100" DestValHigh="100"/>
	<CommCmd Title="6-fach Taster 12345 - Led 2" Comment="" CmdOn="\xFD12345.LED.50.ON.&lt;v&gt;.0\xFE" CmdOff="\xFD12345.LED.50.OFF\xFE" Unit="" Analog="true" Text="false" Sensor="false" SourceValHigh="100" DestValHigh="100"/>
	<CommCmd Title="6-fach Taster 12345 - Led 3" Comment="" CmdOn="\xFD12345.LED.51.ON.&lt;v&gt;.0\xFE" CmdOff="\xFD12345.LED.51.OFF\xFE" Unit="" Analog="true" Text="false" Sensor="false" SourceValHigh="100" DestValHigh="100"/>
	<CommCmd Title="6-fach Taster 12345 - Led 4" Comment="" CmdOn="\xFD12345.LED.52.ON.&lt;v&gt;.0\xFE" CmdOff="\xFD12345.LED.52.OFF\xFE" Unit="" Analog="true" Text="false" Sensor="false" SourceValHigh="100" DestValHigh="100"/>
	<CommCmd Title="6-fach Taster 12345 - Led 5" Comment="" CmdOn="\xFD12345.LED.53.ON.&lt;v&gt;.0\xFE" CmdOff="\xFD12345.LED.53.OFF\xFE" Unit="" Analog="true" Text="false" Sensor="false" SourceValHigh="100" DestValHigh="100"/>
	<CommCmd Title="6-fach Taster 12345 - Led 6" Comment="" CmdOn="\xFD12345.LED.54.ON.&lt;v&gt;.0\xFE" CmdOff="\xFD12345.LED.54.OFF\xFE" Unit="" Analog="true" Text="false" Sensor="false" SourceValHigh="100" DestValHigh="100"/>
	<CommCmd Title="6-fach Taster 12345 - Taster 1" Comment="" CmdOn="\xFD12345.BTN.17.STATUS.\v\xFE" CmdOff="" Unit="&lt;v.x&gt;" Analog="true" Text="false" Sensor="true" SourceValHigh="100" DestValHigh="100"/>
	<CommCmd Title="6-fach Taster 12345 - Taster 2" Comment="" CmdOn="\xFD12345.BTN.18.STATUS.\v\xFE" CmdOff="" Unit="&lt;v.x&gt;" Analog="true" Text="false" Sensor="true" SourceValHigh="100" DestValHigh="100"/>
	<CommCmd Title="6-fach Taster 12345 - Taster 3" Comment="" CmdOn="\xFD12345.BTN.19.STATUS.\v\xFE" CmdOff="" Unit="&lt;v.x&gt;" Analog="true" Text="false" Sensor="true" SourceValHigh="100" DestValHigh="100"/>
	<CommCmd Title="6-fach Taster 12345 - Taster 4" Comment="" CmdOn="\xFD12345.BTN.20.STATUS.\v\xFE" CmdOff="" Unit="&lt;v.x&gt;" Analog="true" Text="false" Sensor="true" SourceValHigh="100" DestValHigh="100"/>
	<CommCmd Title="6-fach Taster 12345 - Taster 5" Comment="" CmdOn="\xFD12345.BTN.21.STATUS.\v\xFE" CmdOff="" Unit="&lt;v.x&gt;" Analog="true" Text="false" Sensor="true" SourceValHigh="100" DestValHigh="100"/>
	<CommCmd Title="6-fach Taster 12345 - Taster 6" Comment="" CmdOn="\xFD12345.BTN.22.STATUS.\v\xFE" CmdOff="" Unit="&lt;v.x&gt;" Analog="true" Text="false" Sensor="true" SourceValHigh="100" DestValHigh="100"/>
	<CommCmd Title="6-fach Taster 12345 - Extern Taster 1" Comment="" CmdOn="\xFD12345.BTN.33.STATUS.\v\xFE" CmdOff="" Unit="&lt;v.x&gt;" Analog="true" Text="false" Sensor="true" SourceValHigh="100" DestValHigh="100"/>
	<CommCmd Title="6-fach Taster 12345 - Extern Taster 2" Comment="" CmdOn="\xFD12345.BTN.34.STATUS.\v\xFE" CmdOff="" Unit="&lt;v.x&gt;" Analog="true" Text="false" Sensor="true" SourceValHigh="100" DestValHigh="100"/>
	<CommCmd Title="6-fach Taster 12345 - Extern Taster 3" Comment="" CmdOn="\xFD12345.BTN.35.STATUS.\v\xFE" CmdOff="" Unit="&lt;v.x&gt;" Analog="true" Text="false" Sensor="true" SourceValHigh="100" DestValHigh="100"/>
	<CommCmd Title="6-fach Taster 12345 - Extern Taster 4" Comment="" CmdOn="\xFD12345.BTN.36.STATUS.\v\xFE" CmdOff="" Unit="&lt;v.x&gt;" Analog="true" Text="false" Sensor="true" SourceValHigh="100" DestValHigh="100"/>
	<CommCmd Title="6-fach Taster 12345 - Extern Taster 5" Comment="" CmdOn="\xFD12345.BTN.37.STATUS.\v\xFE" CmdOff="" Unit="&lt;v.x&gt;" Analog="true" Text="false" Sensor="true" SourceValHigh="100" DestValHigh="100"/>
	<CommCmd Title="6-fach Taster 12345 - Extern Taster 6" Comment="" CmdOn="\xFD12345.BTN.38.STATUS.\v\xFE" CmdOff="" Unit="&lt;v.x&gt;" Analog="true" Text="false" Sensor="true" SourceValHigh="100" DestValHigh="100"/>
	<CommCmd Title="6-fach Taster 12345 - Extern Led 1" Comment="" CmdOn="\xFD12345.LED.65.ON.&lt;v&gt;.0\xFE" CmdOff="\xFD12345.LED.65.OFF\xFE" Unit="" Analog="true" Text="false" Sensor="false" SourceValHigh="100" DestValHigh="100"/>
	<CommCmd Title="6-fach Taster 12345 - Extern Led 2" Comment="" CmdOn="\xFD12345.LED.66.ON.&lt;v&gt;.0\xFE" CmdOff="\xFD12345.LED.66.OFF\xFE" Unit="" Analog="true" Text="false" Sensor="false" SourceValHigh="100" DestValHigh="100"/>
	<CommCmd Title="6-fach Taster 12345 - Extern Led 3" Comment="" CmdOn="\xFD12345.LED.67.ON.&lt;v&gt;.0\xFE" CmdOff="\xFD12345.LED.67.OFF\xFE" Unit="" Analog="true" Text="false" Sensor="false" SourceValHigh="100" DestValHigh="100"/>
	<CommCmd Title="6-fach Taster 12345 - Extern Led 4" Comment="" CmdOn="\xFD12345.LED.68.ON.&lt;v&gt;.0\xFE" CmdOff="\xFD12345.LED.68.OFF\xFE" Unit="" Analog="true" Text="false" Sensor="false" SourceValHigh="100" DestValHigh="100"/>
	<CommCmd Title="6-fach Taster 12345 - Extern Led 5" Comment="" CmdOn="\xFD12345.LED.69.ON.&lt;v&gt;.0\xFE" CmdOff="\xFD12345.LED.69.OFF\xFE" Unit="" Analog="true" Text="false" Sensor="false" SourceValHigh="100" DestValHigh="100"/>
	<CommCmd Title="6-fach Taster 12345 - Extern Led 6" Comment="" CmdOn="\xFD12345.LED.70.ON.&lt;v&gt;.0\xFE" CmdOff="\xFD12345.LED.70.OFF\xFE" Unit="" Analog="true" Text="false" Sensor="false" SourceValHigh="100" DestValHigh="100"/>
	<CommCmd Title="6-fach Taster 12345 - RFID Leser" Comment="" CmdOn="\xFD12345.RFD.65.TAG_ID.\v\xFE" CmdOff="" Unit="&lt;v.x&gt;" Analog="false" Text="true" Sensor="true" SourceValHigh="100" DestValHigh="100"/>
	<CommCmd Title="6-fach Taster 12345 - RFID Leser" Comment="" CmdOn="\xFD12345.RFD.66.TAG_ID.\v\xFE" CmdOff="" Unit="&lt;v.x&gt;" Analog="false" Text="true" Sensor="true" SourceValHigh="100" DestValHigh="100"/>
	<CommCmd Title="6-fach Taster 12345 - RFID Leser" Comment="" CmdOn="\xFD12345.RFD.67.TAG_ID.\v\xFE" CmdOff="" Unit="&lt;v.x&gt;" Analog="false" Text="true" Sensor="true" SourceValHigh="100" DestValHigh="100"/>
	<CommCmd Title="6-fach Taster 12345 - RFID Leser" Comment="" CmdOn="\xFD12345.RFD.68.TAG_ID.\v\xFE" CmdOff="" Unit="&lt;v.x&gt;" Analog="false" Text="true" Sensor="true" SourceValHigh="100" DestValHigh="100"/>
	<CommCmd Title="6-fach Taster 12345 - RFID Leser" Comment="" CmdOn="\xFD12345.RFD.69.TAG_ID.\v\xFE" CmdOff="" Unit="&lt;v.x&gt;" Analog="false" Text="true" Sensor="true" SourceValHigh="100" DestValHigh="100"/>
	</Comm>
*)
END_ACTION

END_FUNCTION_BLOCK

// ---- POUs/RS485_Hausbus_FB/Events/fb_BusTasterEvent.TcPOU
FUNCTION_BLOCK fb_BusTasterEvent
VAR_INPUT
	 I_sID         			:STRING(10);     // Geräte-ID (z.B. '12345')
	 I_sInstID				:STRING(2) 	:=	'17';
	 I_sReceivedString		:STRING(255);	
	 I_bFaultDetection		:BOOL := FALSE;		(* Soll erkennen, ob ein Telegramm für das zurücksetzen eines Tasters nicht gekommen ist *)
	 I_tFaultDetectTime		:TIME := T#10S;
END_VAR
VAR_OUTPUT
	Q_bOut					:BOOL;
END_VAR
VAR
	tonFaultInput			:ton;
	findString0				:STRING ;
	findString1				:STRING ;
END_VAR

(* Automatische Fehlererkennung *)

IF I_bFaultDetection
THEN
	tonFaultInput(
		IN := Q_bOut,
		PT := I_tFaultDetectTime);
END_IF

findString0 := CONCAT(I_sID,'.');
findString0 := CONCAT(findString0,'BTN');
findString0 := CONCAT(findString0,'.');
findString0 := CONCAT(findString0,I_sInstID);
findString0 := CONCAT(findString0,'.');
findString0 := CONCAT(findString0,'STATUS.0');

findString1 := CONCAT(I_sID,'.');
findString1 := CONCAT(findString1,'BTN');
findString1 := CONCAT(findString1,'.');
findString1 := CONCAT(findString1,I_sInstID);
findString1 := CONCAT(findString1,'.');
findString1 := CONCAT(findString1,'STATUS.1');

IF FIND(I_sReceivedString,findString0) >0 
	OR ( tonFaultInput.Q
		AND I_bFaultDetection)
THEN
	Q_bOut := FALSE;
ELSIF
	FIND(I_sReceivedString,findString1) >0 
THEN
	Q_bOut := TRUE;
END_IF

END_FUNCTION_BLOCK

// ---- POUs/RS485_Hausbus_FB/Events/fb_BusTempEvent.TcPOU
FUNCTION_BLOCK fb_BusTempEvent
VAR_INPUT
	 I_sID         			:STRING(10);     // Geräte-ID (z.B. '12345')
	 I_sInstID				:STRING(2) 	:=	'17';
	 I_sReceivedString		:STRING(255);	
	 I_bReset				:BOOL;
	 
END_VAR
VAR_OUTPUT
	Q_lrTemp				:LREAL;
END_VAR
VAR	
	findStringTemp			:STRING;	(* Wird für TMP/ BRS/ RHD verwendet *)

	sTemp1					:STRING;
	sTemp2					:STRING;
	
END_VAR

findStringTemp	:= CONCAT(I_sID,'.');
findStringTemp	:= CONCAT(findStringTemp,'TMP');
findStringTemp	:= CONCAT(findStringTemp,'.');
findStringTemp	:= CONCAT(findStringTemp,I_sInstID);
findStringTemp	:= CONCAT(findStringTemp,'.');

IF I_bReset
THEN
	sTemp1 := '0';
ELSE
	IF FIND(I_sReceivedString,findStringTemp) >0 
	THEN
		sTemp1 :=MID(I_sReceivedString, (* LÄNGE*) 4, FIND(I_sReceivedString,'TMP.1.STATUS.')+ LEN('TMP.1.STATUS.'));
	END_IF
END_IF

Q_lrTemp :=	STRING_TO_LREAL(sTemp1);

END_FUNCTION_BLOCK

// ---- POUs/RS485_Hausbus_FB/Events/fb_BusBrsEvent.TcPOU
FUNCTION_BLOCK fb_BusBrsEvent
VAR_INPUT
	 I_sID         			:STRING(10);     // Geräte-ID (z.B. '12345')
	 I_sInstID				:STRING(2) 	:=	'17';
	 I_sReceivedString		:STRING(255);	
	 I_bReset				:BOOL;
END_VAR
VAR_OUTPUT
	Q_lrBrs				:LREAL;
END_VAR
VAR	
	findStringTemp			:STRING;	(* Wird für TMP/ BRS/ RHD verwendet *)

	sBrs1					:STRING;
	sBrs2					:STRING;
	
END_VAR

findStringTemp	:= CONCAT(I_sID,'.');
findStringTemp	:= CONCAT(findStringTemp,'BRS');
findStringTemp	:= CONCAT(findStringTemp,'.');
findStringTemp	:= CONCAT(findStringTemp,I_sInstID);
findStringTemp	:= CONCAT(findStringTemp,'.');

IF I_bReset
THEN
	sBrs1 := '0';
ELSE
	IF FIND(I_sReceivedString,findStringTemp) >0 
	THEN
		sBrs1 :=MID(I_sReceivedString, (* LÄNGE*) 4, FIND(I_sReceivedString,'BRS.1.STATUS.')+ LEN('BRS.1.STATUS.'));
	END_IF
END_IF

Q_lrBrs :=	STRING_TO_LREAL(sBrs1);

END_FUNCTION_BLOCK

// ---- POUs/RS485_Hausbus_FB/Events/fb_BusRhdEvent.TcPOU
FUNCTION_BLOCK fb_BusRhdEvent
VAR_INPUT
	 I_sID         			:STRING(10);     // Geräte-ID (z.B. '12345')
	 I_sInstID				:STRING(2) 	:=	'17';
	 I_sReceivedString		:STRING(255);	
	 I_bReset				:BOOL;
END_VAR
VAR_OUTPUT
	Q_lrRhd					:LREAL;
END_VAR
VAR	
	findStringTemp			:STRING;	(* Wird für TMP/ BRS/ RHD verwendet *)

	sRhd1					:STRING;
	sRhd2					:STRING;
	
END_VAR

findStringTemp	:= CONCAT(I_sID,'.');
findStringTemp	:= CONCAT(findStringTemp,'RHD');
findStringTemp	:= CONCAT(findStringTemp,'.');
findStringTemp	:= CONCAT(findStringTemp,I_sInstID);
findStringTemp	:= CONCAT(findStringTemp,'.');

IF I_bReset
THEN
	sRhd1 := '0';
ELSE
	IF FIND(I_sReceivedString,findStringTemp) >0 
	THEN
		sRhd1 :=MID(I_sReceivedString, (* LÄNGE*) 4, FIND(I_sReceivedString,'RHD.1.STATUS.')+ LEN('RHD.1.STATUS.'));
	END_IF
END_IF

Q_lrRhd :=	STRING_TO_LREAL(sRhd1);

END_FUNCTION_BLOCK

// ---- POUs/RS485_Hausbus_FB/BusTaster/fb_StringConvTB6F.TcPOU
(*======================================================================================================================================*)
(*fb_StringConvTB6F:	Zusammensetzen des Strings für 6Fach Bust Taster (LEDs und Hintergrundbeleuchtung und Reset)*)
(*
Date          	| Version    	| created under        	| Author          	| Remark *)
(*====================================================================================================================================================*)
(*05/05/2025   	| 1.00      		| TC3		  		| N.Kersting       | first release *)
(*06/05/2025   	| 1.01      		| TC3		  		| N.Kersting       | Externe LEDs Nachgerüstet *)
(*08/05/2025   	| 1.02      		| TC3		  		| N.Kersting       | Umschaltung ob Externe LEDs verwendet werden oder nicht *)
(*====================================================================================================================================================*)
FUNCTION_BLOCK fb_StringConvTB6F
VAR_INPUT
	I_bReset			:BOOL;							(* Reset Befehl auslösen *)
	I_bExtLED			:BOOL;							(* Schaltet nur die Externen LEDs*)
	I_bSetBackground	:BOOL;							(* Nur Hintergrundbeleuchtung setzen *)
	I_bHasExtLED		:BOOL := FALSE;					(* Wenn Aktiv, werden Die Externen LEDs bei Hintergrundbeleuchtung mit gesendet! *)
	I_diID				:DINT;							(* Device ID *)
	I_iLED     	 		:ARRAY[1..6] OF INT;     	  	(* gewünschter LED-Zustand (TRUE = 100 %)*)
	I_iLEDExt  	 		:ARRAY[1..6] OF INT;     	  	(* gewünschter LED-Zustand (TRUE = 100 %)*)
	I_iLEDBg			:INT;							(* gewünschte Hintergrundbeleuchtung Achtung nur für Interne LEDs*)
	I_sStartZeichen		:BYTE := 16#FD;					(* Startzeichen Präfix *)
	I_sEndZeichen		:BYTE := 16#FE;					(* Endzeichen Suffix *)
END_VAR
VAR_OUTPUT
	Q_sConvString		:STRING(255);
END_VAR
VAR
	iStartInstID		:INT :=49;
	iStartLED			:INT := 1;
	
	iStartInstIDExt		:INT :=65;
	iStartLEDExt		:INT := 1;
END_VAR

IF NOT I_bReset
THEN
	IF I_bSetBackground
	THEN
		IF I_bHasExtLED
		THEN
			(* Externe LEDs*)
			iStartInstIDExt := 65;
			iStartLEDExt := 1;
			
			Q_sConvString:=	CONCAT(F_ToCHR(I_sStartZeichen),DINT_TO_STRING(I_diID));
			Q_sConvString:=	CONCAT(Q_sConvString,'.LED.');
			Q_sConvString:=	CONCAT(Q_sConvString,INT_TO_STRING(iStartInstIDExt));
			Q_sConvString:=	CONCAT(Q_sConvString,'.SET_MBR.');
			Q_sConvString:=	CONCAT(Q_sConvString,INT_TO_STRING(I_iLEDBg));
			Q_sConvString:=	CONCAT(Q_sConvString,F_ToCHR(I_sEndZeichen));
			
			iStartInstIDExt := iStartInstIDExt +1;
			iStartLEDExt := 	iStartLEDExt +1;
			
			Q_sConvString:=	CONCAT(Q_sConvString,F_ToCHR(I_sStartZeichen));
			Q_sConvString:=	CONCAT(Q_sConvString,DINT_TO_STRING(I_diID));
			Q_sConvString:=	CONCAT(Q_sConvString,'.LED.');
			Q_sConvString:=	CONCAT(Q_sConvString,INT_TO_STRING(iStartInstIDExt));
			Q_sConvString:=	CONCAT(Q_sConvString,'.SET_MBR.');
			Q_sConvString:=	CONCAT(Q_sConvString,INT_TO_STRING(I_iLEDBg));
			Q_sConvString:=	CONCAT(Q_sConvString,F_ToCHR(I_sEndZeichen));
			
			iStartInstIDExt := iStartInstIDExt +1;
			iStartLEDExt := 	iStartLEDExt +1;
			
			Q_sConvString:=	CONCAT(Q_sConvString,F_ToCHR(I_sStartZeichen));
			Q_sConvString:=	CONCAT(Q_sConvString,DINT_TO_STRING(I_diID));
			Q_sConvString:=	CONCAT(Q_sConvString,'.LED.');
			Q_sConvString:=	CONCAT(Q_sConvString,INT_TO_STRING(iStartInstIDExt));
			Q_sConvString:=	CONCAT(Q_sConvString,'.SET_MBR.');
			Q_sConvString:=	CONCAT(Q_sConvString,INT_TO_STRING(I_iLEDBg));
			Q_sConvString:=	CONCAT(Q_sConvString,F_ToCHR(I_sEndZeichen));
			
			iStartInstIDExt := iStartInstIDExt +1;
			iStartLEDExt := 	iStartLEDExt +1;
			
			Q_sConvString:=	CONCAT(Q_sConvString,F_ToCHR(I_sStartZeichen));
			Q_sConvString:=	CONCAT(Q_sConvString,DINT_TO_STRING(I_diID));
			Q_sConvString:=	CONCAT(Q_sConvString,'.LED.');
			Q_sConvString:=	CONCAT(Q_sConvString,INT_TO_STRING(iStartInstIDExt));
			Q_sConvString:=	CONCAT(Q_sConvString,'.SET_MBR.');
			Q_sConvString:=	CONCAT(Q_sConvString,INT_TO_STRING(I_iLEDBg));
			Q_sConvString:=	CONCAT(Q_sConvString,F_ToCHR(I_sEndZeichen));
			
			iStartInstIDExt := iStartInstIDExt +1;
			iStartLEDExt := 	iStartLEDExt +1;
			
			Q_sConvString:=	CONCAT(Q_sConvString,F_ToCHR(I_sStartZeichen));
			Q_sConvString:=	CONCAT(Q_sConvString,DINT_TO_STRING(I_diID));
			Q_sConvString:=	CONCAT(Q_sConvString,'.LED.');
			Q_sConvString:=	CONCAT(Q_sConvString,INT_TO_STRING(iStartInstIDExt));
			Q_sConvString:=	CONCAT(Q_sConvString,'.SET_MBR.');
			Q_sConvString:=	CONCAT(Q_sConvString,INT_TO_STRING(I_iLEDBg));
			Q_sConvString:=	CONCAT(Q_sConvString,F_ToCHR(I_sEndZeichen));
			
			iStartInstIDExt := iStartInstIDExt +1;
			iStartLEDExt := 	iStartLEDExt +1;
			
			Q_sConvString:=	CONCAT(Q_sConvString,F_ToCHR(I_sStartZeichen));
			Q_sConvString:=	CONCAT(Q_sConvString,DINT_TO_STRING(I_diID));
			Q_sConvString:=	CONCAT(Q_sConvString,'.LED.');
			Q_sConvString:=	CONCAT(Q_sConvString,INT_TO_STRING(iStartInstIDExt));
			Q_sConvString:=	CONCAT(Q_sConvString,'.SET_MBR.');
			Q_sConvString:=	CONCAT(Q_sConvString,INT_TO_STRING(I_iLEDBg));
			Q_sConvString:=	CONCAT(Q_sConvString,F_ToCHR(I_sEndZeichen));
			
			(* Interne LEDs*)
			(* Hintergrundbeleuchtung setzen *)
			
			Q_sConvString:=	CONCAT(Q_sConvString,F_ToCHR(I_sStartZeichen));
			Q_sConvString:=	CONCAT(Q_sConvString,DINT_TO_STRING(I_diID));
			Q_sConvString:=	CONCAT(Q_sConvString,'.LBN.');
			Q_sConvString:=	CONCAT(Q_sConvString,INT_TO_STRING(16));
			Q_sConvString:=	CONCAT(Q_sConvString,'.SET_MBR.');
			Q_sConvString:=	CONCAT(Q_sConvString,INT_TO_STRING(I_iLEDBg));
			Q_sConvString:=	CONCAT(Q_sConvString,F_ToCHR(I_sEndZeichen));
			
		ELSE
			(* Interne LEDs*)
			(* Hintergrundbeleuchtung setzen *)
			Q_sConvString:=	CONCAT(F_ToCHR(I_sStartZeichen),DINT_TO_STRING(I_diID));
			Q_sConvString:=	CONCAT(Q_sConvString,'.LBN.');
			Q_sConvString:=	CONCAT(Q_sConvString,INT_TO_STRING(16));
			Q_sConvString:=	CONCAT(Q_sConvString,'.SET_MBR.');
			Q_sConvString:=	CONCAT(Q_sConvString,INT_TO_STRING(I_iLEDBg));
			Q_sConvString:=	CONCAT(Q_sConvString,F_ToCHR(I_sEndZeichen));
		END_IF
	ELSE
		(* Normale Helligkeit setzen *)
		IF NOT I_bExtLED
		THEN
			(* Interne LEDs*)
			iStartInstID := 49;
			iStartLED := 1;
			
			Q_sConvString:=	CONCAT(F_ToCHR(I_sStartZeichen),DINT_TO_STRING(I_diID));
			Q_sConvString:=	CONCAT(Q_sConvString,'.LED.');
			Q_sConvString:=	CONCAT(Q_sConvString,INT_TO_STRING(iStartInstID));
			Q_sConvString:=	CONCAT(Q_sConvString,'.ON.');
			Q_sConvString:=	CONCAT(Q_sConvString,INT_TO_STRING(I_iLED[iStartLED]));
			Q_sConvString:=	CONCAT(Q_sConvString,F_ToCHR(I_sEndZeichen));
			
			iStartInstID := iStartInstID +1;
			iStartLED := 	iStartLED +1;
			
			Q_sConvString:=	CONCAT(Q_sConvString,F_ToCHR(I_sStartZeichen));
			Q_sConvString:=	CONCAT(Q_sConvString,DINT_TO_STRING(I_diID));
			Q_sConvString:=	CONCAT(Q_sConvString,'.LED.');
			Q_sConvString:=	CONCAT(Q_sConvString,INT_TO_STRING(iStartInstID));
			Q_sConvString:=	CONCAT(Q_sConvString,'.ON.');
			Q_sConvString:=	CONCAT(Q_sConvString,INT_TO_STRING(I_iLED[iStartLED]));
			Q_sConvString:=	CONCAT(Q_sConvString,F_ToCHR(I_sEndZeichen));
			
			iStartInstID := iStartInstID +1;
			iStartLED := 	iStartLED +1;
			
			Q_sConvString:=	CONCAT(Q_sConvString,F_ToCHR(I_sStartZeichen));
			Q_sConvString:=	CONCAT(Q_sConvString,DINT_TO_STRING(I_diID));
			Q_sConvString:=	CONCAT(Q_sConvString,'.LED.');
			Q_sConvString:=	CONCAT(Q_sConvString,INT_TO_STRING(iStartInstID));
			Q_sConvString:=	CONCAT(Q_sConvString,'.ON.');
			Q_sConvString:=	CONCAT(Q_sConvString,INT_TO_STRING(I_iLED[iStartLED]));
			Q_sConvString:=	CONCAT(Q_sConvString,F_ToCHR(I_sEndZeichen));
			
			iStartInstID := iStartInstID +1;
			iStartLED := 	iStartLED +1;
			
			Q_sConvString:=	CONCAT(Q_sConvString,F_ToCHR(I_sStartZeichen));
			Q_sConvString:=	CONCAT(Q_sConvString,DINT_TO_STRING(I_diID));
			Q_sConvString:=	CONCAT(Q_sConvString,'.LED.');
			Q_sConvString:=	CONCAT(Q_sConvString,INT_TO_STRING(iStartInstID));
			Q_sConvString:=	CONCAT(Q_sConvString,'.ON.');
			Q_sConvString:=	CONCAT(Q_sConvString,INT_TO_STRING(I_iLED[iStartLED]));
			Q_sConvString:=	CONCAT(Q_sConvString,F_ToCHR(I_sEndZeichen));
			
			iStartInstID := iStartInstID +1;
			iStartLED := 	iStartLED +1;
			
			Q_sConvString:=	CONCAT(Q_sConvString,F_ToCHR(I_sStartZeichen));
			Q_sConvString:=	CONCAT(Q_sConvString,DINT_TO_STRING(I_diID));
			Q_sConvString:=	CONCAT(Q_sConvString,'.LED.');
			Q_sConvString:=	CONCAT(Q_sConvString,INT_TO_STRING(iStartInstID));
			Q_sConvString:=	CONCAT(Q_sConvString,'.ON.');
			Q_sConvString:=	CONCAT(Q_sConvString,INT_TO_STRING(I_iLED[iStartLED]));
			Q_sConvString:=	CONCAT(Q_sConvString,F_ToCHR(I_sEndZeichen));
			
